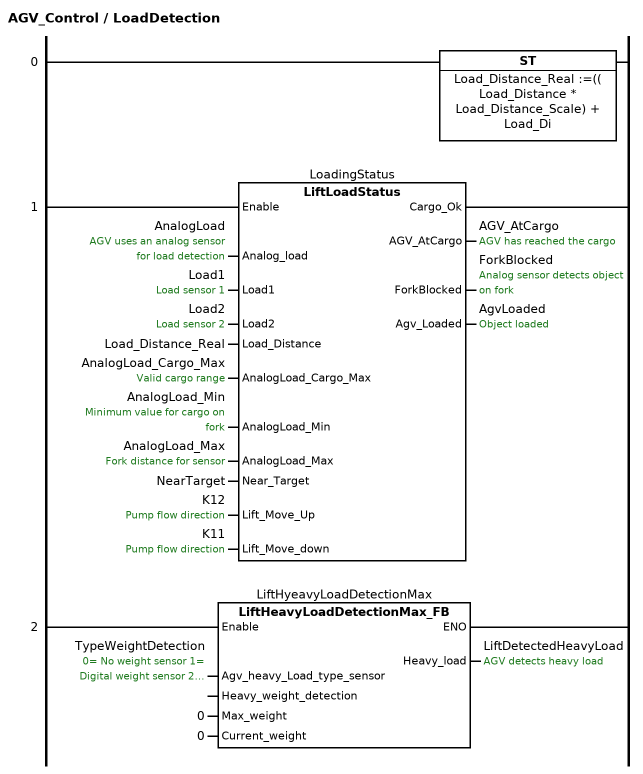
(* Rung 0 *)
Load_Distance_Real :=(( Load_Distance * Load_Distance_Scale) + Load_Distance_Offset);
(* Rung 1 *)
LoadingStatus(Enable := TRUE, Analog_load := AnalogLoad, Load1 := Load1, Load2 := Load2, Load_Distance := Load_Distance_Real, AnalogLoad_Cargo_Max := AnalogLoad_Cargo_Max, AnalogLoad_Min := AnalogLoad_Min, AnalogLoad_Max := AnalogLoad_Max, Near_Target := NearTarget, Lift_Move_Up := K12, Lift_Move_down := K11, AGV_AtCargo => AGV_AtCargo, ForkBlocked => ForkBlocked, Agv_Loaded => AgvLoaded);
(* Rung 2 *)
LiftHyeavyLoadDetectionMax(Enable := TRUE, Agv_heavy_Load_type_sensor := TypeWeightDetection, Max_weight := 0, Current_weight := 0, Heavy_load => LiftDetectedHeavyLoad);

(* Section Bufferlane: ladder, written here as Structured Text *)

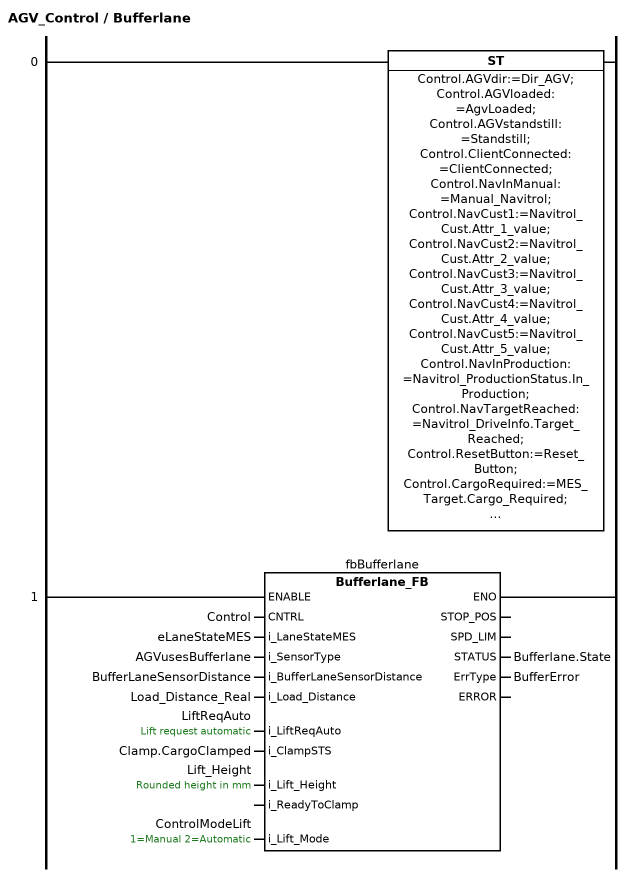
(* Rung 0 *)
Control.AGVdir:=Dir_AGV;
Control.AGVloaded:=AgvLoaded;
Control.AGVstandstill:=Standstill;
Control.ClientConnected:=ClientConnected;
Control.NavInManual:=Manual_Navitrol;
Control.NavCust1:=Navitrol_Cust.Attr_1_value;
Control.NavCust2:=Navitrol_Cust.Attr_2_value;
Control.NavCust3:=Navitrol_Cust.Attr_3_value;
Control.NavCust4:=Navitrol_Cust.Attr_4_value;
Control.NavCust5:=Navitrol_Cust.Attr_5_value;
Control.NavInProduction:=Navitrol_ProductionStatus.In_Production;
Control.NavTargetReached:=Navitrol_DriveInfo.Target_Reached;
Control.ResetButton:=Reset_Button;
Control.CargoRequired:=MES_Target.Cargo_Required;

MES_LanePickState:=Bufferlane.State.ePickSTAT;
MES_LaneDropState:=Bufferlane.State.eDropSTAT;
(* Rung 1 *)
fbBufferlane(ENABLE := TRUE, CNTRL := Control, i_LaneStateMES := eLaneStateMES, i_SensorType := AGVusesBufferlane, i_BufferLaneSensorDistance := BufferLaneSensorDistance, i_Load_Distance := Load_Distance_Real, i_LiftReqAuto := LiftReqAuto, i_ClampSTS := Clamp.CargoClamped, i_Lift_Height := Lift_Height, i_Lift_Mode := ControlModeLift, STATUS => Bufferlane.State, ErrType => BufferError);
END_PROGRAM

PROGRAM Communication
VAR
    Host : STRING[256];
    ServerPort : INT;
    Willconfig_Mqtt : MQTT\WillCnfg;
    mqttbuffer : MQTT\ClientBuffer;
    mqttclient : MQTT\MQTTClient;
    start_up : TON;
    mqttping : MQTT\MQTTPing;
    rcv_message : STRING[1986];
    rcv_topic : STRING[128];
    mqttsub : MQTT\MQTTSubscribe;
    rcv_message_mes : STRING[1986];
    rcv_topic_mes : STRING[128];
    mqttsub_mes : MQTT\MQTTSubscribe;
    rcv_message_target : STRING[1986];
    rcv_topic_target : STRING[128];
    mqttsub_target : MQTT\MQTTSubscribe;
    sendRequest : BOOL;
    mqttpublish : MQTT\MQTTPublish;
    pub_topic : STRING[128];
    act_topic : STRING[128];  (* MQTT topic for actuator commands from MES *)
    pub_message : STRING[1986];
    act_message : STRING[1986];  (* MQTT message for responding to actuator commands *)
    pub_i : UINT;
END_VAR
VAR RETAIN
    machid : STRING[20];
END_VAR
VAR
    SerialSetupDone : BOOL;  (* RS232 setup state done *)
    RS_TX_Done : BOOL;  (* Serial buffer send *)
    debug_receiveserial : BOOL;
    debug_sendserial : BOOL;
    SendSerial1 : BOOL;  (* Send serial message 1 *)
    SerialTimer_PT : TIME;  (* Cycle time *)
    SerialTimer_ET : TIME;  (* Elapsed time *)
    SerialTimer_TON : TON;
    RS_Clear_Done : BOOL;  (* Serial buffer cleared *)
    DevicePort : _sDEVICE_PORT;  (* RS232 port *)
    SerialSendDat : ARRAY[0..4] OF BYTE;  (* TX byte array *)
    SerialSendSize : UINT;  (* Amount of bytes to send *)
    SerialSendConfig : _sSERIAL_CFG;  (* Block config *)
    SerialSendOption : _sSERIAL_SEND_OPTION;  (* Transmission option *)
    RS_Abort : BOOL;  (* Halt serial communication *)
    RS_TX_Busy : BOOL;  (* Transmission in progress *)
    RS_TX_Aborted : BOOL;  (* Transmission has been aborted *)
    RS_TX_Error : BOOL;  (* Error active in serial send *)
    RS_TX_ErrorID : WORD;  (* Error ID *)
    RS232_TX : NX_SerialSend;  (* Send serial data *)
    RS_RX_Done : BOOL;  (* Serial buffer read *)
    SerialReceive : ARRAY[0..49] OF BYTE;  (* Serial message in Bytes *)
    SerialRecvSize : UINT;  (* Amount of bytes we want to read *)
    SerialRcvConfig : _sSERIAL_CFG;  (* block config *)
    SerialRcvOption : _sSERIAL_RCV_OPTION;  (* Transmission option *)
    RS_RS_Busy : BOOL;  (* Read in progress *)
    RS_RX_Aborted : BOOL;  (* Read has been aborted *)
    RS_RX_Error : BOOL;  (* Error active in serial read *)
    RS_RX_ErrorID : WORD;  (* Error ID *)
    RS_RX_Size : UINT;  (* Amount of bytes read *)
    RS232_RX : NX_SerialRcv;  (* Receive serial data from buffer *)
    debug_clearserial : BOOL;
    RS232_Clear_Busy : BOOL;  (* Buffer clearing in pogress *)
    RS232_Clear : NX_SerialBufClear;  (* Serial RXbuffer clear *)
    HandleSerialData : BOOL;  (* Apply filters and calculate distance *)
    ReceivedChecksum : BYTE;  (* Last received XOR checksum *)
    SerialOk : BOOL;  (* Checksum ok on received data *)
    SerialDataSaved : BOOL;  (* All distances and echos received ok *)
    Distances : ARRAY[0..10] OF UINT;  (* All distances from RS232 sensor *)
    Echos : ARRAY[0..10] OF UINT;  (* All echos from RS232 sensor *)
    FirstUpdateDone : BOOL;  (* Serial data has been received *)
    OverhangDetected : BOOL;  (* Overhead detection measurements within limit *)
    Overhang_ChargerOverride : BOOL;  (* AGV is aproaching the charger *)
    Overhang_PT : TIME;  (* time an object must be within bounds *)
    Overhang_ET : TIME;  (* Elapsed time *)
    Overhang_TON : TON;  (* Overhang stability timer *)
    Checksum : BYTE;  (* Calculated checksum *)
    IndexCheck : UINT;  (* index for checksum calculation *)
    NrOfBeams : UINT;  (* Amount of beams per scan *)
    Xserial : ARRAY[0..10] OF INT;  (* Calculated X values from measurements *)
    Angle : ARRAY[0..10] OF REAL;  (* Angles in radians *)
    Yserial : ARRAY[0..10] OF INT;  (* Calculated Y values from measurements *)
    IndexLimit : UINT;
    Ylimit : INT;  (* Distance the RS232 beams are allowed to go sideways *)
    Xlimit : INT;  (* Distance the RS232 beams should be able to reach towards the front *)
    PublishIndex : INT;
    MqttActRequest : BOOL;  (* Transmit update *)
    mqtt_target_publish : MQTT\MQTTPublish;
    mqttsub_palletDetection : MQTT\MQTTSubscribe;
    palletDetection_topic : STRING[128];
    rcv_message_palletDetection : STRING[1986];
    rcv_topic_palletDetection : STRING[128];
    Mqtt_client_ID : STRING[128];
    error_topic : STRING[128];
    HMI_IP_Init : BOOL;
    Host_Block1 : STRING[18];
    Host_Block2 : STRING[18];
    mqtt_test_done : BOOL;
    mqttsub_error : MQTT\MQTTSubscribe;
    mqttsub_popup : MQTT\MQTTSubscribe;
    mqttsub_warning : MQTT\MQTTSubscribe;
    popup_topic : STRING[128];
    rcv_message_error : STRING[1986];
    rcv_message_popup : STRING[1986];
    rcv_message_warning : STRING[1986];
    rcv_popup_info : STRING[128];
    rcv_topic_error : STRING[128];
    rcv_topic_warning : STRING[128];
    warning_topic : STRING[128];
    mqttsub_language : MQTT\MQTTSubscribe;
    language_topic : STRING[128];
    laneDropStateMES_topic : STRING[128];
    laneStateMES_topic : STRING[128];
    mqttsub_laneStateMES : MQTT\MQTTSubscribe;
    mqttsub_MES_BufferState : MQTT\MQTTSubscribe;
    rcv_message_laneDropStateMES : STRING[1986];
    rcv_message_laneStateMES : STRING[128];
    rcv_topic_laneDropStateMES : STRING[128];
    rcv_topic_laneStateMES : STRING[128];
END_VAR
VAR_EXTERNAL
    ClientConnected : BOOL;
    Mqtt_values : ARRAY[0..32] OF MQTTval;
    Stations_State : Node_State;
    MES_State : Node_State;
    MES_Target : MQTT_Actuator_Request_struct;
    AGVusesRS232 : BOOL;
    AGV_Init : UINT;
    Dir_Encoder1 : BOOL;
    Brake_Override_Switch : BOOL;
    Manual_ControlModeLift : BOOL;
    AGV_Docking : BOOL;
    Reset_Flag : BOOL;
    Navitrol_Tag : Navitrol_Status_TagV4_sec_struct;
    ToChargerTag : UDINT;
    ChargerTag : UDINT;
    Standstill : BOOL;
    Charge_Relay : BOOL;
END_VAR
VAR_EXTERNAL CONSTANT
    RS232_BoardID : _sOPTBOARD_ID;
END_VAR
VAR_EXTERNAL
    MachineID : INT;
    Warning_Mqtt_Client_Error : BOOL;
    MQTT_enabled : BOOL;  (* MES communication type enabled *)
    MES_PalletDetection : Palletdetection_Action;
    OptionalFieldReq : INT;
    RS232_OverhangDetected : BOOL;
    HMI_Int12 : INT;
    HMI_Int13 : INT;
    HMI_Int14 : INT;
    HMI_Int15 : INT;
    IP_Block1 : INT;
    IP_Block2 : INT;
    IP_Block3 : INT;
    IP_Block4 : INT;
    MES_Error : MQTT_Errors_struct;
    MES_Popup : MQTT_Popup_struct;
    MES_Warning : MQTT_Warnings_struct;
    HMI_Input13 : BOOL;
    HMI_Int16 : INT;
    MES_Language : INT;
    eLaneStateMES : Lane_state_MES;
    Manual_Mode : BOOL;
END_VAR
VAR
    _p1 : BOOL;
    _e2 : R_TRIG;
    _e3 : R_TRIG;
    _e4 : R_TRIG;
    _e5 : R_TRIG;
    _p6 : BOOL;
    _p7 : BOOL;
END_VAR

(* Section Client: ladder, written here as Structured Text *)

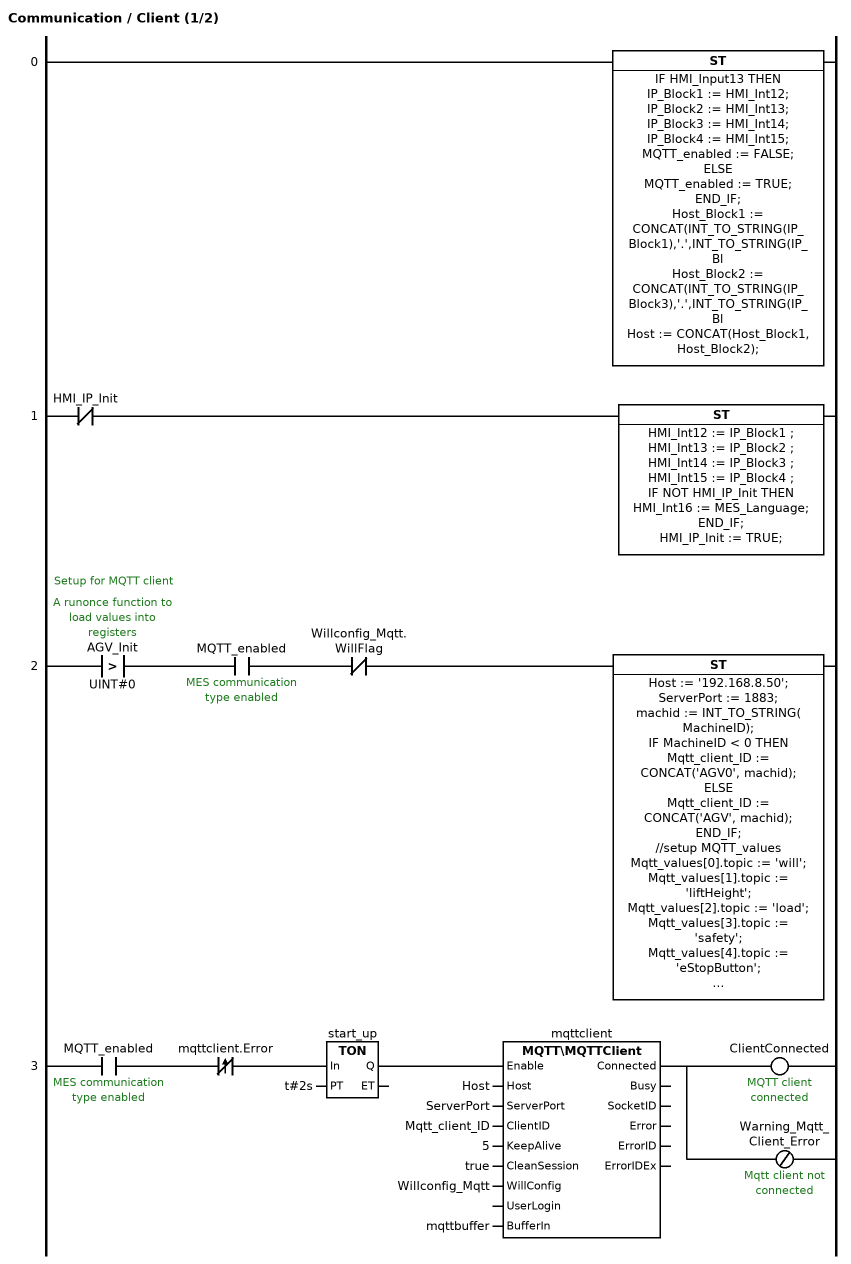
(* Rung 0 *)
IF HMI_Input13 THEN
	IP_Block1 := HMI_Int12;
	IP_Block2 := HMI_Int13;
	IP_Block3 := HMI_Int14;
	IP_Block4 := HMI_Int15;

	MQTT_enabled := FALSE;
	
ELSE
	MQTT_enabled := TRUE;
END_IF;

Host_Block1 := CONCAT(INT_TO_STRING(IP_Block1),'.',INT_TO_STRING(IP_Block2),'.');
Host_Block2 := CONCAT(INT_TO_STRING(IP_Block3),'.',INT_TO_STRING(IP_Block4));
Host := CONCAT(Host_Block1,Host_Block2);
(* Rung 1 *)
_p1 := NOT HMI_IP_Init;
IF _p1 THEN
    HMI_Int12 := IP_Block1 ;
    HMI_Int13 := IP_Block2 ;
    HMI_Int14 := IP_Block3 ;
    HMI_Int15 := IP_Block4 ;
    
    IF NOT HMI_IP_Init THEN
    	HMI_Int16 := MES_Language;
    END_IF;
    
    HMI_IP_Init := TRUE;
END_IF;
(* Rung 2: Setup for MQTT client *)
IF (AGV_Init > UINT#0) AND MQTT_enabled AND NOT Willconfig_Mqtt.WillFlag THEN
    Host := '192.168.8.50';
    ServerPort := 1883;
    machid := INT_TO_STRING(MachineID);
    IF MachineID < 0 THEN
    	Mqtt_client_ID := CONCAT('AGV0', machid);
    ELSE
    	Mqtt_client_ID := CONCAT('AGV', machid);
    END_IF;
    
    //setup MQTT_values
    Mqtt_values[0].topic := 'will';
    Mqtt_values[1].topic := 'liftHeight';
    Mqtt_values[2].topic := 'load';
    Mqtt_values[3].topic := 'safety';
    Mqtt_values[4].topic := 'eStopButton';
    Mqtt_values[5].topic := 'scanner1';
    Mqtt_values[6].topic := 'scanner2';
    Mqtt_values[7].topic := 'palletDetection/state';
    Mqtt_values[8].topic := 'docking';
    Mqtt_values[9].topic := 'manualDrive';
    Mqtt_values[10].topic := 'manualLift';
    Mqtt_values[11].topic := 'brakeRelease';
    Mqtt_values[12].topic := 'charging';
    Mqtt_values[13].topic := 'cancelRequest';
    Mqtt_values[14].topic := 'cancelConfirm';
    Mqtt_values[15].topic := 'forkCollision';
    Mqtt_values[16].topic := 'palletDetection/countedPallets';
    Mqtt_values[17].topic := 'heavyLoad';
    Mqtt_values[18].topic := 'laneDropStateAGV';
    Mqtt_values[19].topic := 'palletDetection';
    Mqtt_values[20].topic := 'errorsWarnings';
    Mqtt_values[21].topic := 'palletDetectionAngle';
    Mqtt_values[22].topic := 'popUp/operatorConfirmation';
    Mqtt_values[23].topic := 'popUp/operatorCancelation';
    Mqtt_values[24].topic := 'language';
    Mqtt_values[25].topic := 'lanePickStateAGV';
    
    //config for firstrun. required for startup
    Willconfig_Mqtt.WillTopic :=  CONCAT('agvs/',machid,'/will');
    Willconfig_Mqtt.WillMsg := 'Offline';
    Willconfig_Mqtt.WillRetain := TRUE;
    Willconfig_Mqtt.WillQoS := 0;
    Willconfig_Mqtt.WillFlag := TRUE;
    
    //Actuator values
    act_topic := CONCAT('agvs/',INT_TO_STRING(MachineID),'/target');
    palletDetection_topic := CONCAT('agvs/',INT_TO_STRING(MachineID),'/palletDetection/active');
    popup_topic:=CONCAT('agvs/',INT_TO_STRING(MachineID),'/popUp');
    language_topic:=CONCAT('agvs/',INT_TO_STRING(MachineID),'/language');
    laneStateMES_topic:=CONCAT('agvs/',INT_TO_STRING(MachineID),'/laneActionStateMES');
END_IF;
(* Rung 3 *)
_e2(CLK := mqttclient.Error);
start_up(In := MQTT_enabled AND NOT _e2.Q, PT := t#2s);
mqttclient(Enable := start_up.Q, Host := Host, ServerPort := ServerPort, ClientID := Mqtt_client_ID, KeepAlive := 5, CleanSession := true, WillConfig := Willconfig_Mqtt, BufferIn := mqttbuffer);
ClientConnected := mqttclient.Connected;
Warning_Mqtt_Client_Error := NOT mqttclient.Connected;

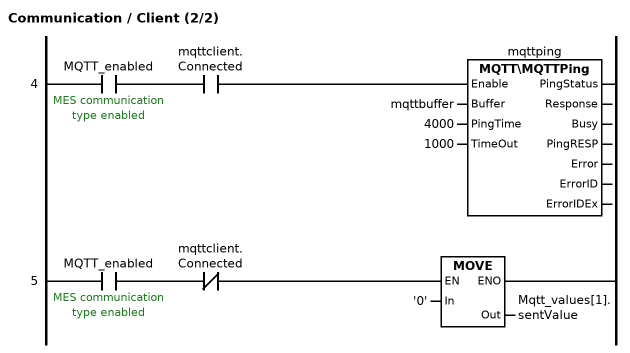
(* Rung 4 *)
mqttping(Enable := MQTT_enabled AND mqttclient.Connected, Buffer := mqttbuffer, PingTime := 4000, TimeOut := 1000);
(* Rung 5 *)
IF MQTT_enabled AND NOT mqttclient.Connected THEN Mqtt_values[1].sentValue := '0'; END_IF;

(* Section Subscribe: ladder, written here as Structured Text *)

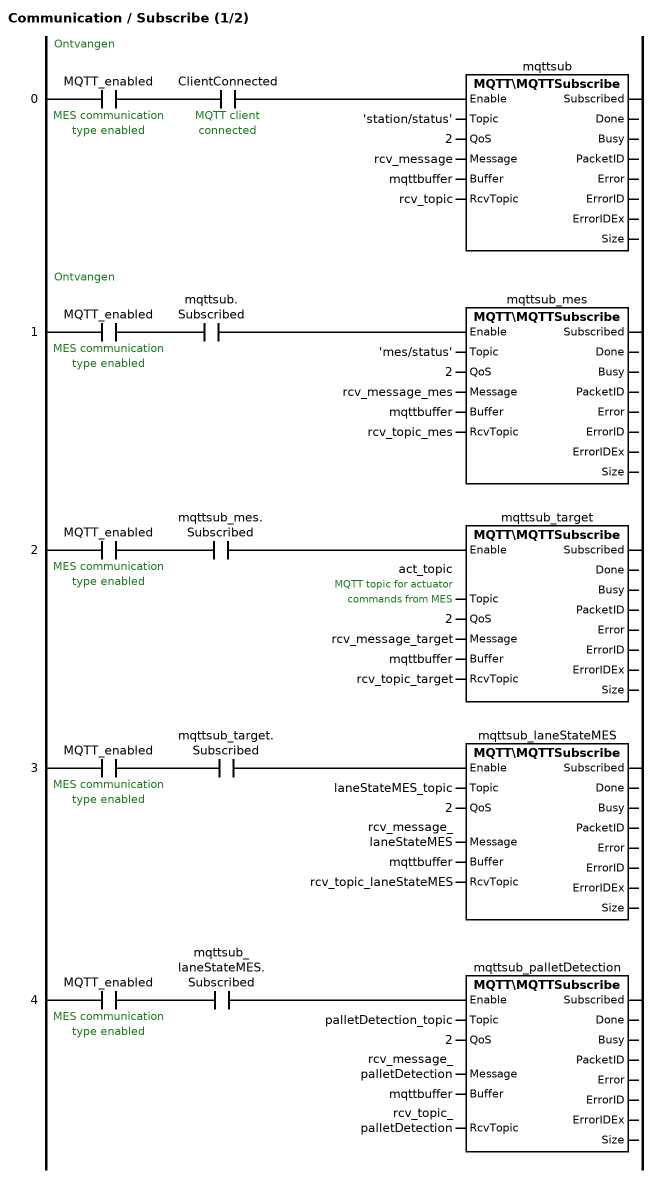
(* Rung 0: Ontvangen *)
mqttsub(Enable := MQTT_enabled AND ClientConnected, Topic := 'station/status', QoS := 2, Message := rcv_message, Buffer := mqttbuffer, RcvTopic := rcv_topic);
(* Rung 1: Ontvangen *)
mqttsub_mes(Enable := MQTT_enabled AND mqttsub.Subscribed, Topic := 'mes/status', QoS := 2, Message := rcv_message_mes, Buffer := mqttbuffer, RcvTopic := rcv_topic_mes);
(* Rung 2 *)
mqttsub_target(Enable := MQTT_enabled AND mqttsub_mes.Subscribed, Topic := act_topic, QoS := 2, Message := rcv_message_target, Buffer := mqttbuffer, RcvTopic := rcv_topic_target);
(* Rung 3 *)
mqttsub_laneStateMES(Enable := MQTT_enabled AND mqttsub_target.Subscribed, Topic := laneStateMES_topic, QoS := 2, Message := rcv_message_laneStateMES, Buffer := mqttbuffer, RcvTopic := rcv_topic_laneStateMES);
(* Rung 4 *)
mqttsub_palletDetection(Enable := MQTT_enabled AND mqttsub_laneStateMES.Subscribed, Topic := palletDetection_topic, QoS := 2, Message := rcv_message_palletDetection, Buffer := mqttbuffer, RcvTopic := rcv_topic_palletDetection);

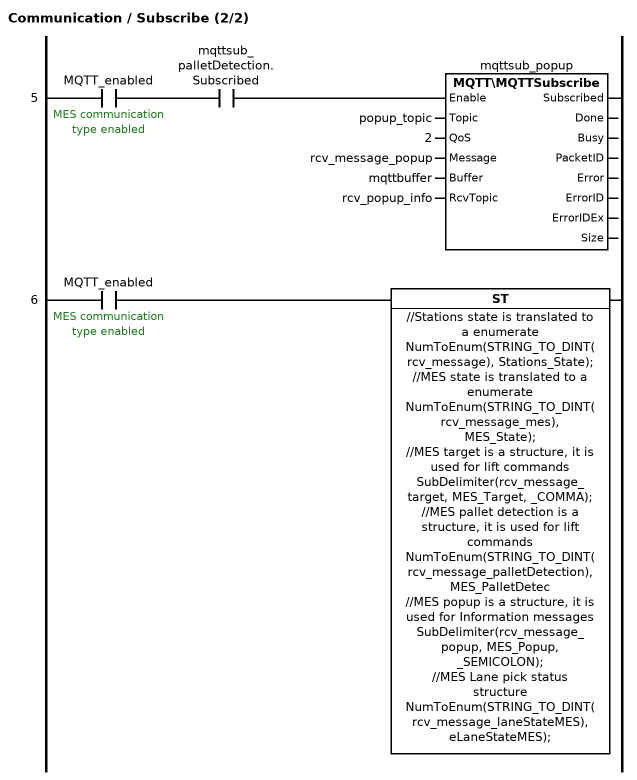
(* Rung 5 *)
mqttsub_popup(Enable := MQTT_enabled AND mqttsub_palletDetection.Subscribed, Topic := popup_topic, QoS := 2, Message := rcv_message_popup, Buffer := mqttbuffer, RcvTopic := rcv_popup_info);
(* Rung 6 *)
IF MQTT_enabled THEN
    //Stations state is translated to a enumerate
    NumToEnum(STRING_TO_DINT(rcv_message), Stations_State);
    //MES state is translated to a enumerate
    NumToEnum(STRING_TO_DINT(rcv_message_mes), MES_State);
    //MES target is a structure, it is used for lift commands
    SubDelimiter(rcv_message_target, MES_Target, _COMMA);
    //MES pallet detection is a structure, it is used for lift commands
    NumToEnum(STRING_TO_DINT(rcv_message_palletDetection), MES_PalletDetection);
    //MES popup is a structure, it is used for Information messages
    SubDelimiter(rcv_message_popup, MES_Popup, _SEMICOLON);
    //MES Lane pick status structure
    NumToEnum(STRING_TO_DINT(rcv_message_laneStateMES), eLaneStateMES);
END_IF;

(* Section Publish: ladder, written here as Structured Text *)

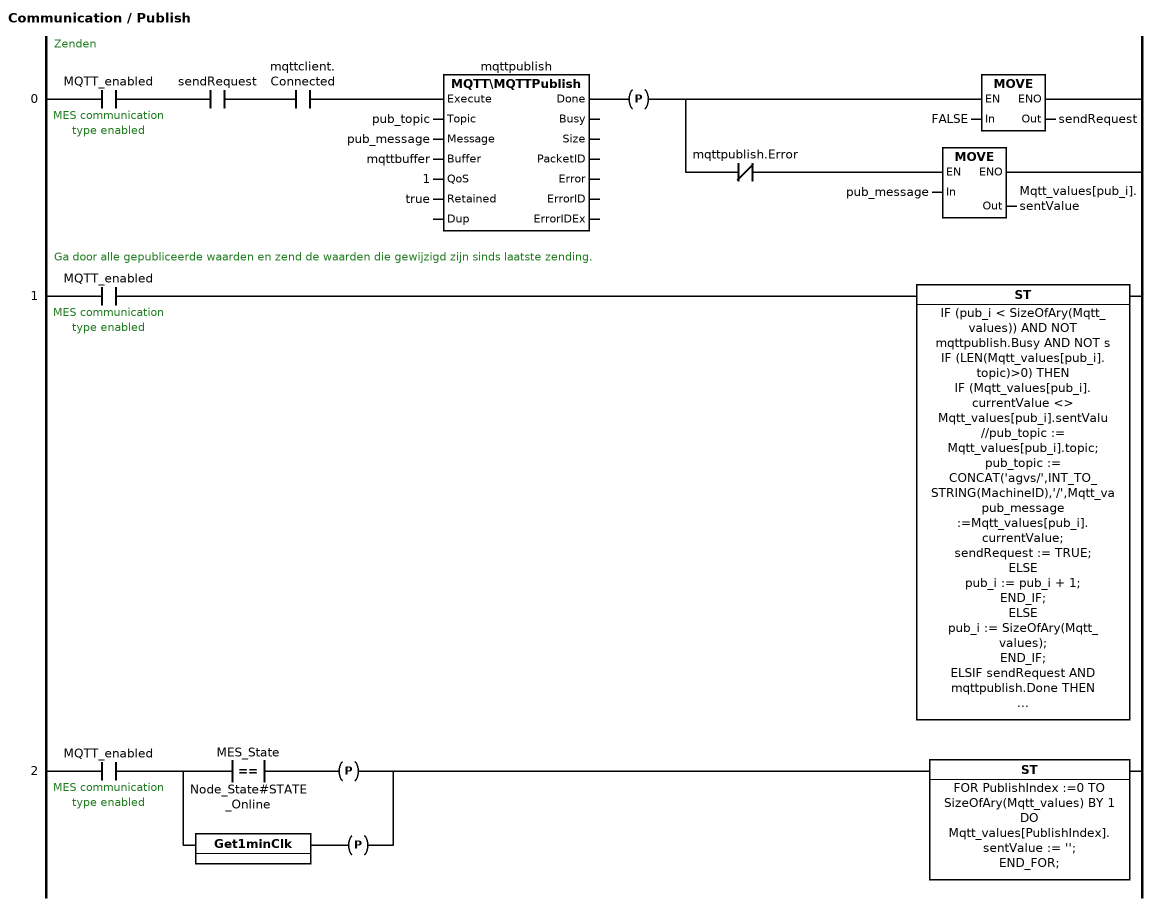
(* Rung 0: Zenden *)
mqttpublish(Execute := MQTT_enabled AND sendRequest AND mqttclient.Connected, Topic := pub_topic, Message := pub_message, Buffer := mqttbuffer, QoS := 1, Retained := true);
_e3(CLK := mqttpublish.Done);
IF _e3.Q THEN sendRequest := FALSE; END_IF;
IF _e3.Q AND NOT mqttpublish.Error THEN Mqtt_values[pub_i].sentValue := pub_message; END_IF;
(* Rung 1: Ga door alle gepubliceerde waarden en zend de waarden die gewijzigd zijn sinds laatste zending. *)
IF MQTT_enabled THEN
    IF (pub_i < SizeOfAry(Mqtt_values)) AND NOT mqttpublish.Busy AND NOT sendRequest THEN
    	IF (LEN(Mqtt_values[pub_i].topic)>0) THEN
    		IF (Mqtt_values[pub_i].currentValue <> Mqtt_values[pub_i].sentValue ) THEN
    			//pub_topic := Mqtt_values[pub_i].topic;
    			pub_topic := CONCAT('agvs/',INT_TO_STRING(MachineID),'/',Mqtt_values[pub_i].topic);
    			pub_message :=Mqtt_values[pub_i].currentValue;
    			sendRequest := TRUE;
    		ELSE
    		pub_i := pub_i + 1;
    		END_IF;
    	ELSE
    		pub_i := SizeOfAry(Mqtt_values);
    	END_IF;
    ELSIF sendRequest AND mqttpublish.Done THEN
    	sendRequest := FALSE;
    	Mqtt_values[pub_i].sentValue := pub_message;
    END_IF;
    IF (pub_i >= SizeOfAry(Mqtt_values)) THEN
    	pub_i := 0;
    END_IF;
END_IF;
(* Rung 2 *)
_e4(CLK := MQTT_enabled AND (MES_State = Node_State#STATE_Online));
_e5(CLK := MQTT_enabled AND Get1minClk());
IF _e4.Q OR _e5.Q THEN
    FOR PublishIndex :=0 TO SizeOfAry(Mqtt_values) BY 1 DO
    	Mqtt_values[PublishIndex].sentValue := '';
    END_FOR;
END_IF;

(* Section RS232: ladder, written here as Structured Text *)

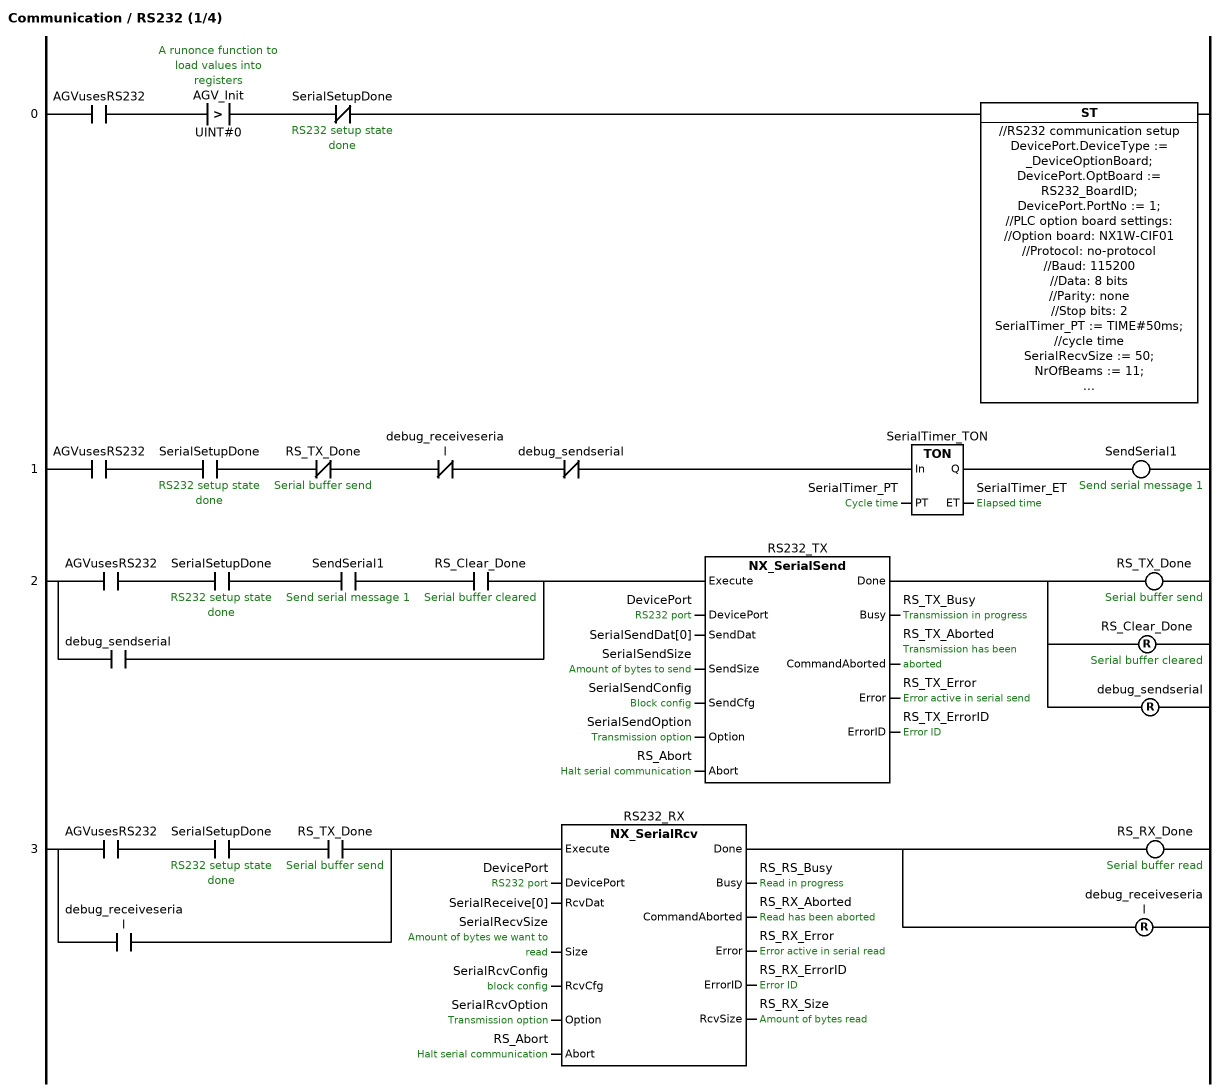
(* Rung 0 *)
IF AGVusesRS232 AND (AGV_Init > UINT#0) AND NOT SerialSetupDone THEN
    //RS232 communication setup
    DevicePort.DeviceType := _DeviceOptionBoard;
    DevicePort.OptBoard := RS232_BoardID;
    DevicePort.PortNo := 1;
    
    //PLC option board settings:
    //Option board: NX1W-CIF01
    //Protocol: no-protocol
    //Baud: 115200
    //Data: 8 bits
    //Parity: none
    //Stop bits: 2
    
    SerialTimer_PT := TIME#50ms;	//cycle time
    SerialRecvSize := 50;
    NrOfBeams := 11;
    Ylimit := 600; //distance in mm
    Xlimit := 2000; //distance in mm
    Overhang_PT := TIME#100ms;  //time an object must be in limit area until waring becomes active
    
    //TX settings
    SerialSendSize := 5;							//we send 5 bytes in total
    SerialSendOption.SendDelay := 0;	//minimal delay in transmission
    
    //Fill (Default) TX data
    SerialSendDat[0] := BYTE#222;	//0xDE = sender
    SerialSendDat[1] := BYTE#1;		//0x01 = receiver
    SerialSendDat[2] := BYTE#5;		//0x05 = amount of bytes
    SerialSendDat[3] := BYTE#89;	//0x59 = command (read)
    SerialSendDat[4] := BYTE#131;	//0x83 = XOR checksum
    
    //fill angle per beam (lookup table)
    Angle[0] := DegToRad(REAL#40);
    Angle[1] := DegToRad(REAL#32);
    Angle[2] := DegToRad(REAL#24);
    Angle[3] := DegToRad(REAL#16);
    Angle[4] := DegToRad(REAL#8);
    Angle[5] := DegToRad(REAL#0);
    Angle[6] := DegToRad(REAL#8);
    Angle[7] := DegToRad(REAL#16);
    Angle[8] := DegToRad(REAL#24);
    Angle[9] := DegToRad(REAL#32);
    Angle[10] := DegToRad(REAL#40);
    
    SerialSetupDone := TRUE;
    RS_Clear_Done := TRUE;
END_IF;
(* Rung 1 *)
SerialTimer_TON(In := AGVusesRS232 AND SerialSetupDone AND NOT RS_TX_Done AND NOT debug_receiveserial AND NOT debug_sendserial, PT := SerialTimer_PT, ET => SerialTimer_ET);
SendSerial1 := SerialTimer_TON.Q;
(* Rung 2 *)
RS232_TX(Execute := (AGVusesRS232 AND SerialSetupDone AND SendSerial1 AND RS_Clear_Done) OR debug_sendserial, DevicePort := DevicePort, SendDat := SerialSendDat[0], SendSize := SerialSendSize, SendCfg := SerialSendConfig, Option := SerialSendOption, Abort := RS_Abort, Busy => RS_TX_Busy, CommandAborted => RS_TX_Aborted, Error => RS_TX_Error, ErrorID => RS_TX_ErrorID);
RS_TX_Done := RS232_TX.Done;
IF RS232_TX.Done THEN
    RS_Clear_Done := FALSE;
    debug_sendserial := FALSE;
END_IF;
(* Rung 3 *)
RS232_RX(Execute := (AGVusesRS232 AND SerialSetupDone AND RS_TX_Done) OR debug_receiveserial, DevicePort := DevicePort, RcvDat := SerialReceive[0], Size := SerialRecvSize, RcvCfg := SerialRcvConfig, Option := SerialRcvOption, Abort := RS_Abort, Busy => RS_RS_Busy, CommandAborted => RS_RX_Aborted, Error => RS_RX_Error, ErrorID => RS_RX_ErrorID, RcvSize => RS_RX_Size);
RS_RX_Done := RS232_RX.Done;
IF RS232_RX.Done THEN debug_receiveserial := FALSE; END_IF;

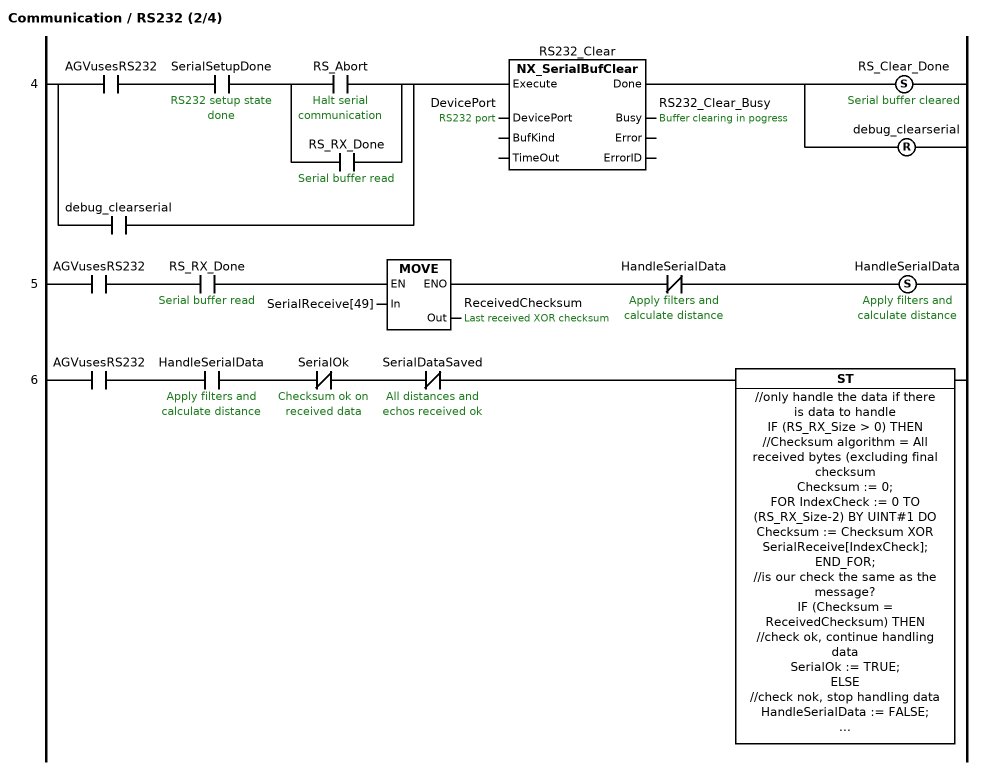
(* Rung 4 *)
RS232_Clear(Execute := (AGVusesRS232 AND SerialSetupDone AND (RS_Abort OR RS_RX_Done)) OR debug_clearserial, DevicePort := DevicePort, Busy => RS232_Clear_Busy);
IF RS232_Clear.Done THEN
    RS_Clear_Done := TRUE;
    debug_clearserial := FALSE;
END_IF;
(* Rung 5 *)
IF AGVusesRS232 AND RS_RX_Done THEN ReceivedChecksum := SerialReceive[49]; END_IF;
IF AGVusesRS232 AND RS_RX_Done AND NOT HandleSerialData THEN HandleSerialData := TRUE; END_IF;
(* Rung 6 *)
_p6 := AGVusesRS232 AND HandleSerialData AND NOT SerialOk AND NOT SerialDataSaved;
IF _p6 THEN
    //only handle the data if there is data to handle
    IF (RS_RX_Size > 0) THEN
    	//Checksum algorithm = All received bytes (excluding final checksum byte) must be XOR
    	Checksum := 0;
    	FOR IndexCheck := 0 TO (RS_RX_Size-2) BY UINT#1 DO
    		Checksum := Checksum XOR SerialReceive[IndexCheck];
    	END_FOR;
    	//is our check the same as the message?
    	IF (Checksum = ReceivedChecksum) THEN
    		//check ok, continue handling data
    		SerialOk := TRUE;
    	ELSE
    		//check nok, stop handling data
    		HandleSerialData := FALSE;
    	END_IF;
    ELSE
    	//no data, stop handling data
    	HandleSerialData := FALSE;
    END_IF;
    	
END_IF;

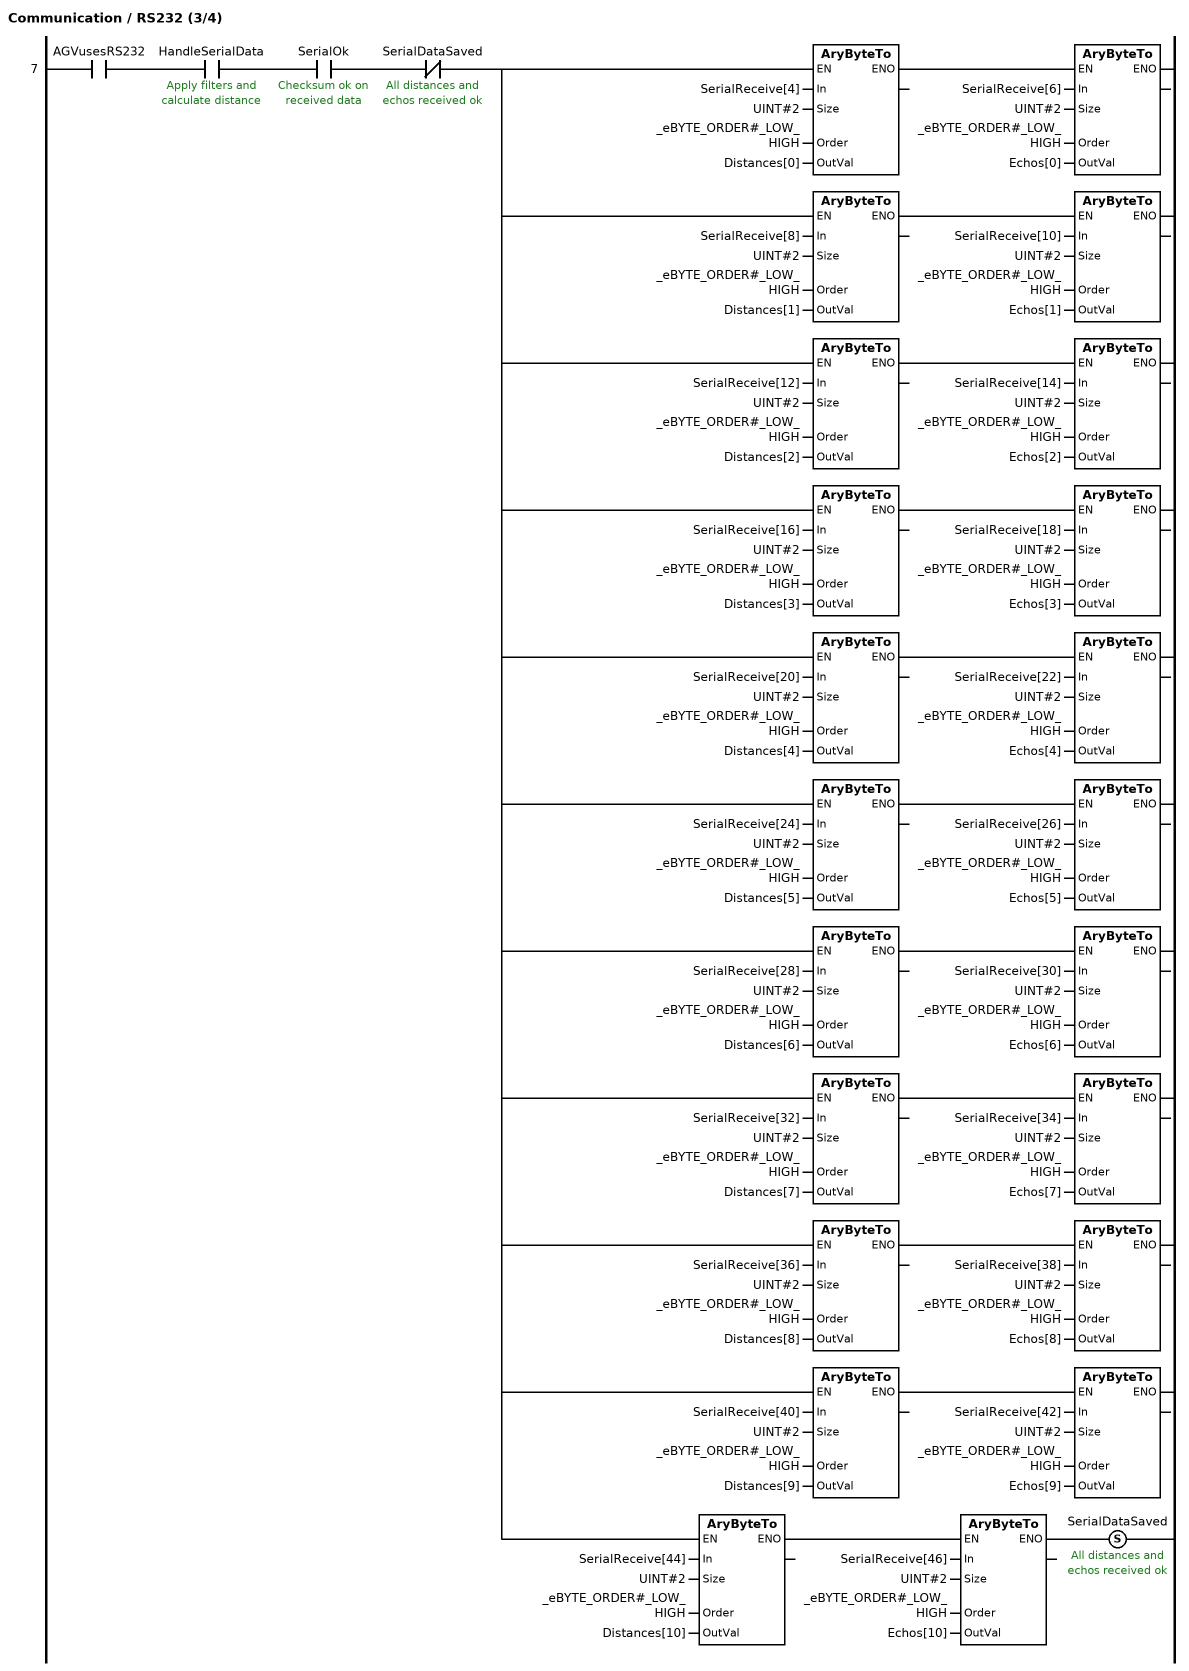
(* Rung 7 *)
_p7 := AGVusesRS232 AND HandleSerialData AND SerialOk AND NOT SerialDataSaved;
IF _p7 THEN
    AryByteTo(In := SerialReceive[4], Size := UINT#2, Order := _eBYTE_ORDER#_LOW_HIGH, OutVal := Distances[0]);
    AryByteTo(In := SerialReceive[6], Size := UINT#2, Order := _eBYTE_ORDER#_LOW_HIGH, OutVal := Echos[0]);
    AryByteTo(In := SerialReceive[8], Size := UINT#2, Order := _eBYTE_ORDER#_LOW_HIGH, OutVal := Distances[1]);
    AryByteTo(In := SerialReceive[10], Size := UINT#2, Order := _eBYTE_ORDER#_LOW_HIGH, OutVal := Echos[1]);
    AryByteTo(In := SerialReceive[12], Size := UINT#2, Order := _eBYTE_ORDER#_LOW_HIGH, OutVal := Distances[2]);
    AryByteTo(In := SerialReceive[14], Size := UINT#2, Order := _eBYTE_ORDER#_LOW_HIGH, OutVal := Echos[2]);
    AryByteTo(In := SerialReceive[16], Size := UINT#2, Order := _eBYTE_ORDER#_LOW_HIGH, OutVal := Distances[3]);
    AryByteTo(In := SerialReceive[18], Size := UINT#2, Order := _eBYTE_ORDER#_LOW_HIGH, OutVal := Echos[3]);
    AryByteTo(In := SerialReceive[20], Size := UINT#2, Order := _eBYTE_ORDER#_LOW_HIGH, OutVal := Distances[4]);
    AryByteTo(In := SerialReceive[22], Size := UINT#2, Order := _eBYTE_ORDER#_LOW_HIGH, OutVal := Echos[4]);
    AryByteTo(In := SerialReceive[24], Size := UINT#2, Order := _eBYTE_ORDER#_LOW_HIGH, OutVal := Distances[5]);
    AryByteTo(In := SerialReceive[26], Size := UINT#2, Order := _eBYTE_ORDER#_LOW_HIGH, OutVal := Echos[5]);
    AryByteTo(In := SerialReceive[28], Size := UINT#2, Order := _eBYTE_ORDER#_LOW_HIGH, OutVal := Distances[6]);
    AryByteTo(In := SerialReceive[30], Size := UINT#2, Order := _eBYTE_ORDER#_LOW_HIGH, OutVal := Echos[6]);
    AryByteTo(In := SerialReceive[32], Size := UINT#2, Order := _eBYTE_ORDER#_LOW_HIGH, OutVal := Distances[7]);
    AryByteTo(In := SerialReceive[34], Size := UINT#2, Order := _eBYTE_ORDER#_LOW_HIGH, OutVal := Echos[7]);
    AryByteTo(In := SerialReceive[36], Size := UINT#2, Order := _eBYTE_ORDER#_LOW_HIGH, OutVal := Distances[8]);
    AryByteTo(In := SerialReceive[38], Size := UINT#2, Order := _eBYTE_ORDER#_LOW_HIGH, OutVal := Echos[8]);
    AryByteTo(In := SerialReceive[40], Size := UINT#2, Order := _eBYTE_ORDER#_LOW_HIGH, OutVal := Distances[9]);
    AryByteTo(In := SerialReceive[42], Size := UINT#2, Order := _eBYTE_ORDER#_LOW_HIGH, OutVal := Echos[9]);
    AryByteTo(In := SerialReceive[44], Size := UINT#2, Order := _eBYTE_ORDER#_LOW_HIGH, OutVal := Distances[10]);
    AryByteTo(In := SerialReceive[46], Size := UINT#2, Order := _eBYTE_ORDER#_LOW_HIGH, OutVal := Echos[10]);
    SerialDataSaved := TRUE;
END_IF;

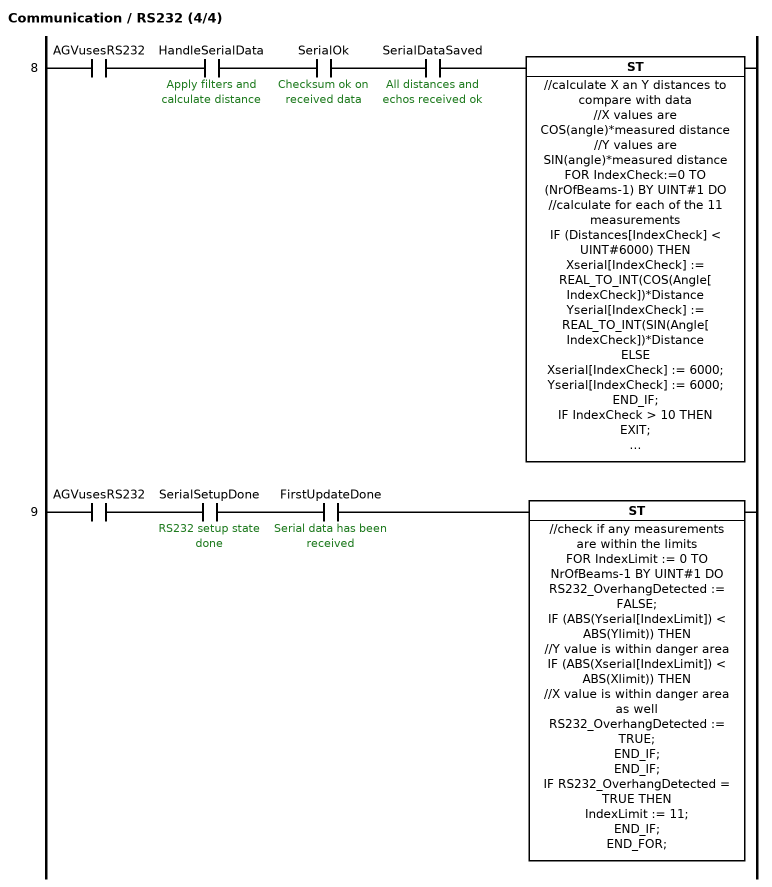
(* Rung 8 *)
IF AGVusesRS232 AND HandleSerialData AND SerialOk AND SerialDataSaved THEN
    //calculate X an Y distances to compare with data
    //X values are COS(angle)*measured distance
    //Y values are SIN(angle)*measured distance
    FOR IndexCheck:=0 TO (NrOfBeams-1) BY UINT#1 DO
    	//calculate for each of the 11 measurements
    	IF (Distances[IndexCheck] < UINT#6000) THEN
    		Xserial[IndexCheck] := REAL_TO_INT(COS(Angle[IndexCheck])*Distances[IndexCheck]);
    		Yserial[IndexCheck] := REAL_TO_INT(SIN(Angle[IndexCheck])*Distances[IndexCheck]);
    	ELSE
    		Xserial[IndexCheck] := 6000;
    		Yserial[IndexCheck] := 6000;
    	END_IF;
    	IF IndexCheck > 10 THEN
    		EXIT;
    	END_IF;
    END_FOR;
    
    //Checks done
    SerialDataSaved := FALSE;
    SerialOk := FALSE;
    HandleSerialData := FALSE;
    FirstUpdateDone := TRUE;
END_IF;
(* Rung 9 *)
IF AGVusesRS232 AND SerialSetupDone AND FirstUpdateDone THEN
    //check if any measurements are within the limits
    FOR IndexLimit := 0 TO NrOfBeams-1 BY UINT#1 DO
    	RS232_OverhangDetected := FALSE;
    	IF (ABS(Yserial[IndexLimit]) < ABS(Ylimit)) THEN
    		//Y value is within danger area
    		IF (ABS(Xserial[IndexLimit]) < ABS(Xlimit)) THEN
    			//X value is within danger area as well
    			RS232_OverhangDetected := TRUE;
    		END_IF;
    	END_IF;
    	IF RS232_OverhangDetected = TRUE THEN
    		IndexLimit := 11;
    	END_IF;
    END_FOR;
END_IF;
END_PROGRAM

PROGRAM Manual_control
VAR
    AnalogFwdRevInput : INT := 0;  (* Combined input from both F/R channels *)
END_VAR
VAR CONSTANT
    CenterCounts : INT := 1000;  (* 2,5V on -4000/4000 counts *)
    AnalogMaxFwdCounts : INT := 2000;  (* Maximum counts when joystick max forward *)
    AnalogMaxLeftCounts : INT := 0;  (* Maximum counts when joystick max left *)
    AnalogMaxRevCounts : INT := 0000;  (* Minimum counts when joystick max reverse *)
    AnalogMaxRightCounts : INT := 2000;  (* Minimum counts when joystick max right *)
END_VAR
VAR
    PercentFwdRev : INT := 0;  (* Percentage in forward/reverse (-100=max rev, 100 = max fwd) *)
    PercentLeftRight : INT := 0;  (* Percentage in left/right (-100=max left, 100=max right) *)
    AnalogLeftRightInput : INT := 0;
    RM_FR1Avg : INT := 0;  (* Average value of RM_FR1 channel *)
    alpha : INT := 10;  (* alpha = between 0 and 100, for averaging *)
    RM_LR1Avg : INT := 0;  (* Average value of RM_LR1 channel *)
    RM_CenterAvg : INT := 0;  (* Average value of RM_Center channel *)
    ManualConnect : SktTCPConnect;
    ManualSocket : _sSOCKET;
    ManualSend : SktTCPSend;
    payload : ARRAY[0..150] OF BYTE := [16#50,16#4f,16#53,16#54,16#20,16#2f,16#72,16#65,16#6d,16#6f,16#74,16#65,16#5f,16#63,16#6f,16#6e,16#74,16#72,16#6f,16#6c,16#3f,16#78,16#3d,16#30,16#2e,16#30,16#30,16#30,16#26,16#79,16#3d,16#30,16#2e,16#30,16#30,16#30,16#26,16#74,16#65,16#61,16#63,16#68,16#3d,16#30,16#26,16#6d,16#61,16#6e,16#75,16#61,16#6c,16#3d,16#31,16#26,16#66,16#61,16#73,16#74,16#3d,16#31,16#26,16#67,16#65,16#74,16#5f,16#63,16#6f,16#6e,16#74,16#72,16#6f,16#6c,16#3d,16#30,16#26,16#6f,16#6d,16#6e,16#69,16#5f,16#74,16#79,16#70,16#65,16#3d,16#32,16#26,16#6f,16#6d,16#6e,16#69,16#5f,16#66,16#6f,16#72,16#77,16#3d,16#31,16#20,16#48,16#54,16#54,16#50,16#2f,16#31,16#2e,16#31,16#0d,16#0a,16#48,16#6f,16#73,16#74,16#3a,16#20,16#31,16#39,16#32,16#2e,16#31,16#36,16#38,16#2e,16#31,16#32,16#37,16#2e,16#31,16#0d,16#0a,16#43,16#6f,16#6e,16#74,16#65,16#6e,16#74,16#2d,16#4c,16#65,16#6e,16#67,16#74,16#68,16#3a,16#20,16#30,16#0d,16#0a,16#0d,16#0a];
    WebPayload : ARRAY[0..250] OF BYTE;
    ASCII : ARRAY[0..9] OF BYTE := [16#30, 16#31, 16#32, 16#33, 16#34, 16#35, 16#36, 16#37, 16#38, 16#39];
    X_ABS : USINT;
    Y_ABS : USINT;
    ManualDisconnect : SktClose;
    ManualConnected : BOOL;  (* Connection to Navitrol made *)
    Sendsize : UINT;  (* amount of bytes to send *)
    Manual_Init : INT;  (* run once *)
    ManualRecv : SktTCPRcv;
    Recv_Payload : ARRAY[0..999] OF BYTE;
    Recv_Bytes : UINT;  (* Amount of bytes from buffer *)
    Got_Manual : BOOL;  (* received data *)
    Recv_String : STRING[500];
    Data_Index : UINT;
    TestByte : BYTE;
    Data_Start : STRING[9];
    debug_ButtonPressed : BOOL;
    Byte_Order : _eBYTE_ORDER := _LOW_HIGH;
    Result : UINT;
    String_Input : STRING[24];
    Got_Manual_String : BOOL;  (* Collected data *)
    Web_Feedback : Webinterface_Reply_struct;
    PLC_IP : STRING[15] := '192.168.127.2';
    debug_NEascii : BOOL;
    debug_EQascii : BOOL;
    GetToken0 : GetToken;
    TestToken : ARRAY[0..4] OF BYTE;
    Manual_Clk : BOOL;  (* debug variable *)
    Process_Manual_String : BOOL;  (* Data ready for handling *)
    Recv_Data : STRING[500];
    ManualStatus : SktGetTCPStatus;
    ManualSocket_Status : _eCONNECTION_STATE;  (* status at last send *)
    Skt_State_Closed : _eCONNECTION_STATE := _CLOSED;
    ManualClearBuffer : SktClearBuf;
    KeepAliveTON : TON;
    Keepalive_PT : TIME := 150ms;  (* time until connection is reset *)
    Keepalive_ET : TIME;  (* elapsed time *)
    ManualDisconnect0 : SktClose;
    ManualConnect0 : SktTCPConnect;
    ManualReconnect : BOOL;
    ResetAliveTON : TON;
    Skt_State_Closing : _eCONNECTION_STATE := _CLOSE_WAIT;
    String_Index : INT;
    ResetTON : TON;
    Manual_Reset_PT : TIME := 250ms;  (* time for reset *)
    Manual_Reset_ET : TIME;
    ManualTOF : TOF;
    KeepOff_PT : TIME := 50ms;  (* Reset time *)
    KeepOff_ET : TIME;  (* elapsed time *)
    GetToken1 : GetToken;
    GetToken2 : GetToken;
END_VAR
VAR_EXTERNAL
    RM_FR1 : INT;
    RM_Center : INT;
    RM_LR1 : INT;
    IPC_Driving_active : BOOL;
    IPC_Driving_x : INT;
    IPC_Driving_y : INT;
    RM_Switch : INT;
    Manual_ControlModeLift : BOOL;  (* Switch or HMI manual *)
    RemoteButtonPressed : BOOL;  (* Joystick button is pressed *)
    AGVhasHandheld : BOOL;
    Navitrol_status : Navitrol_Status_Struct;
    RM_Dwn : INT;
    RM_Up : INT;
    Remote_Present : BOOL;  (* Remote present and ok *)
    HMI_Input10 : BOOL;
    Rm_ManUp : BOOL;
    Rm_ManDown : BOOL;
    Error_Remote : BOOL;  (* Center tap voltage too low, no remote connected *)
    Navitrol_gen : Navitrol_Status_General_Sec_Struct;
    Update_Navitrol : BOOL;
    AGV_Init : UINT;
    Charge_Relay : BOOL;
    TCPReady : BOOL;
    Manual_Mode : BOOL;  (* Switch or HMI manual *)
END_VAR
VAR
    _e1 : R_TRIG;
    _e2 : F_TRIG;
    _e3 : R_TRIG;
    _p4 : BOOL;
    _e5 : R_TRIG;
    _e6 : F_TRIG;
    _e7 : R_TRIG;
    _e8 : F_TRIG;
    _e9 : F_TRIG;
    _p10 : BOOL;
    _p11 : BOOL;
    _p12 : BOOL;
    _p13 : BOOL;
END_VAR

(* Section ManualControl: ladder, written here as Structured Text *)

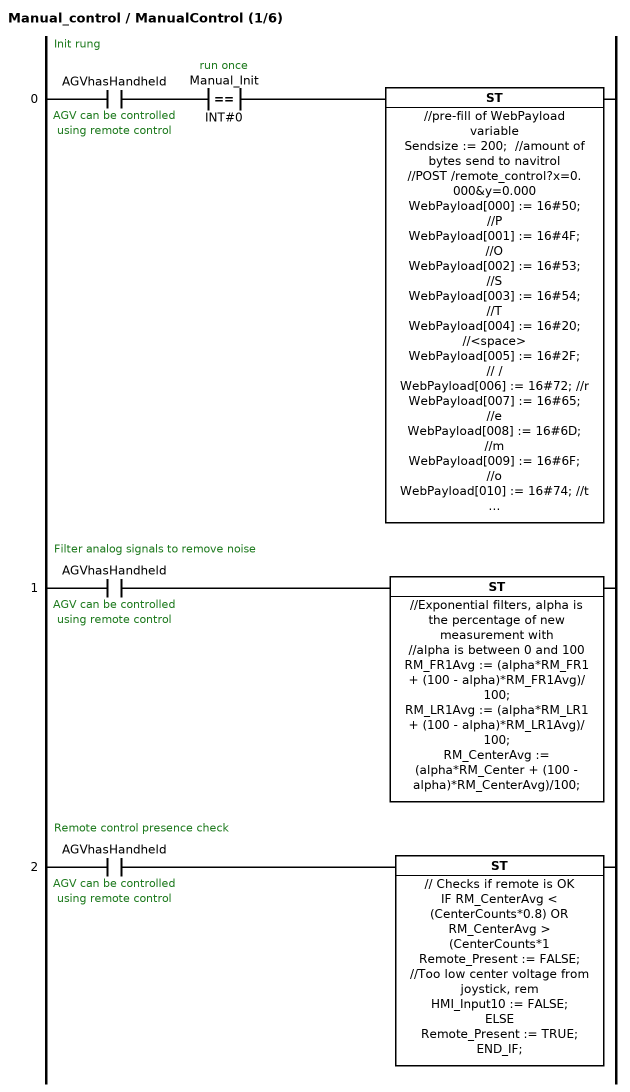
(* Rung 0: Init rung *)
IF AGVhasHandheld AND (Manual_Init = INT#0) THEN
    //pre-fill of WebPayload variable
    Sendsize := 200;	//amount of bytes send to navitrol
    //POST /remote_control?x=0.000&y=0.000
    WebPayload[000] := 16#50;	//P
    WebPayload[001] := 16#4F;		//O
    WebPayload[002] := 16#53;	//S
    WebPayload[003] := 16#54;	//T
    WebPayload[004] := 16#20;	//<space>
    WebPayload[005] := 16#2F;		// /
    WebPayload[006] := 16#72;	//r
    WebPayload[007] := 16#65;	//e
    WebPayload[008] := 16#6D;	//m
    WebPayload[009] := 16#6F;		//o
    WebPayload[010] := 16#74;	//t
    WebPayload[011] := 16#65;	//e
    WebPayload[012] := 16#5F;		//_
    WebPayload[013] := 16#63;	//c
    WebPayload[014] := 16#6F;		//o
    WebPayload[015] := 16#6E;	//n
    WebPayload[016] := 16#74;	//t
    WebPayload[017] := 16#72;	//r
    WebPayload[018] := 16#6F;		//o
    WebPayload[019] := 16#6C;	//l
    WebPayload[020] := 16#3F;		//?
    WebPayload[021] := 16#78;	//x
    WebPayload[022] := 16#3D;	//=
    WebPayload[023] := ASCII[0];	//joystick value (4 bytes)
    WebPayload[024] := 16#2E;	//.
    WebPayload[025] := ASCII[0];	//0
    WebPayload[026] := ASCII[0];	//0
    WebPayload[027] := ASCII[0];	//0
    WebPayload[028] := 16#26;	//&
    WebPayload[029] := 16#79;	//y
    WebPayload[030] := 16#3D;	//=
    WebPayload[031] := ASCII[0];	//joystick value (4 bytes)
    WebPayload[032] := 16#2E;	//.
    WebPayload[033] := ASCII[0];	//0
    WebPayload[034] := ASCII[0];	//0
    WebPayload[035] := ASCII[0];	//0
    //&teach=0
    WebPayload[036] := 16#26;	//&
    WebPayload[037] := 16#74;	//t
    WebPayload[038] := 16#65;	//e
    WebPayload[039] := 16#61;	//a
    WebPayload[040] := 16#63;	//c
    WebPayload[041] := 16#68;	//h
    WebPayload[042] := 16#3D;	//=
    WebPayload[043] := ASCII[0];	//teach ControlModeLift on/off (1 byte)
    //&manual=1
    WebPayload[044] := 16#26;	//&
    WebPayload[045] := 16#6D;	//m
    WebPayload[046] := 16#61;	//a
    WebPayload[047] := 16#6E;	//n
    WebPayload[048] := 16#75;	//u
    WebPayload[049] := 16#61;	//a
    WebPayload[050] := 16#6C;	//l
    WebPayload[051] := 16#3D;	//=
    WebPayload[052] := ASCII[0];	//manual control on/off (1 byte)
    //&fast=0
    WebPayload[053] := 16#26;	//&
    WebPayload[054] := 16#66;	//f
    WebPayload[055] := 16#61;	//a
    WebPayload[056] := 16#73;	//s
    WebPayload[057] := 16#74;	//t
    WebPayload[058] := 16#3D;	//=
    WebPayload[059] := ASCII[0];	//unkown value (1 byte)
    //&get_control=0
    WebPayload[060] := 16#26;	//&
    WebPayload[061] := 16#67;	//g
    WebPayload[062] := 16#65;	//e
    WebPayload[063] := 16#74;	//t
    WebPayload[064] := 16#5F;		//_
    WebPayload[065] := 16#63;	//c
    WebPayload[066] := 16#6F;		//o
    WebPayload[067] := 16#6E;	//n
    WebPayload[068] := 16#74;	//t
    WebPayload[069] := 16#72;	//r
    WebPayload[070] := 16#6F;		//o
    WebPayload[071] := 16#6C;	//l
    WebPayload[072] := 16#3D;	//=
    WebPayload[073] := ASCII[0];	//request to be controller (1 byte)
    //&omni_type=2
    WebPayload[074] := 16#26;	//&
    WebPayload[075] := 16#6F;		//o
    WebPayload[076] := 16#6D;	//m
    WebPayload[077] := 16#6E;	//n
    WebPayload[078] := 16#69;	//i
    WebPayload[079] := 16#5F;		//_
    WebPayload[080] := 16#74;	//t
    WebPayload[081] := 16#79;	//y
    WebPayload[082] := 16#70;	//p
    WebPayload[083] := 16#65;	//e
    WebPayload[084] := 16#3D;	//=
    WebPayload[085] := ASCII[2];	//unkown value (1 byte)
    //&omni_forw=1
    WebPayload[086] := 16#26;	//&
    WebPayload[087] := 16#6F;		//o
    WebPayload[088] := 16#6D;	//m
    WebPayload[089] := 16#6E;	//n
    WebPayload[090] := 16#69;	//i
    WebPayload[091] := 16#5F;		//_
    WebPayload[092] := 16#66;	//f
    WebPayload[093] := 16#6F;		//o
    WebPayload[094] := 16#72;	//r
    WebPayload[095] := 16#77;	//w
    WebPayload[096] := 16#3D;	//=
    WebPayload[097] := ASCII[1];	//unknown value (1 byte)
    //&token=00000
    WebPayload[098] := 16#26;	//&
    WebPayload[099] := 16#74;	//t
    WebPayload[100] := 16#6F;		//o
    WebPayload[101] := 16#6B;	//k
    WebPayload[102] := 16#65;	//e
    WebPayload[103] := 16#6E;	//n
    WebPayload[104] := 16#3D;	//=
    WebPayload[105] := ASCII[0];	//identifier (5 bytes)
    WebPayload[106] := ASCII[0];	//0
    WebPayload[107] := ASCII[0];	//0
    WebPayload[108] := ASCII[0];	//0
    WebPayload[109] := ASCII[0];	//0
    //&loadunload=0
    WebPayload[110] := 16#26;	//&
    WebPayload[111] := 16#6C;	//l
    WebPayload[112] := 16#6F;		//o
    WebPayload[113] := 16#61;	//a
    WebPayload[114] := 16#64;	//d
    WebPayload[115] := 16#75;	//u
    WebPayload[116] := 16#6E;	//n
    WebPayload[117] := 16#6C;	//l
    WebPayload[118] := 16#6F;		//o
    WebPayload[119] := 16#61;	//a
    WebPayload[120] := 16#64;	//d
    WebPayload[121] := 16#3D;	//=
    WebPayload[122] := ASCII[0];	//0
    //<space>HTTP/1.1<cr><nl>
    WebPayload[123] := 16#20;	//<space>
    WebPayload[124] := 16#48;	//H
    WebPayload[125] := 16#54;	//T
    WebPayload[126] := 16#54;	//T
    WebPayload[127] := 16#50;	//P
    WebPayload[128] := 16#2F	;	// /
    WebPayload[129] := ASCII[1];	//1
    WebPayload[130] := 16#2E;	//.
    WebPayload[131] := ASCII[1];	//1
    WebPayload[132] := 16#0D;	//<cr>
    WebPayload[133] := 16#0A;	//<nl>
    //Host:<space>192.168.127.1<cr><nl>
    WebPayload[134] := 16#48;	//H
    WebPayload[135] := 16#6F;		//o
    WebPayload[136] := 16#73;	//s
    WebPayload[137] := 16#74;	//t
    WebPayload[138] := 16#3A;	//:
    WebPayload[139] := 16#20;	//<space>
    WebPayload[140] := ASCII[1];	//1
    WebPayload[141] := ASCII[9];	//9
    WebPayload[142] := ASCII[2];	//2
    WebPayload[143] := 16#2E;	//.
    WebPayload[144] := ASCII[1];	//1
    WebPayload[145] := ASCII[6];	//6
    WebPayload[146] := ASCII[8];	//8
    WebPayload[147] := 16#2E;	//.
    WebPayload[148] := ASCII[1];	//1
    WebPayload[149] := ASCII[2];	//2
    WebPayload[150] := ASCII[7];	//7
    WebPayload[151] := 16#2E;	//.
    WebPayload[152] := ASCII[1];	//1
    WebPayload[153] := 16#0D;	//<cr>
    WebPayload[154] := 16#0A;	//<nl>
    //Connection:<space>keep-alive<cr><nl>
    WebPayload[155] := 16#43;	//C
    WebPayload[156] := 16#6F;		//o
    WebPayload[157] := 16#6E;	//n
    WebPayload[158] := 16#6E;	//n
    WebPayload[159] := 16#65;	//e
    WebPayload[160] := 16#63;	//c
    WebPayload[161] := 16#74;	//t
    WebPayload[162] := 16#69;	//i
    WebPayload[163] := 16#6F;		//o
    WebPayload[164] := 16#6E;	//n
    WebPayload[165] := 16#3A;	//:
    WebPayload[166] := 16#20;	//<space>
    WebPayload[167] := 16#6B;	//k
    WebPayload[168] := 16#65;	//e
    WebPayload[169] := 16#65;	//e
    WebPayload[170] := 16#70;	//p
    WebPayload[171] := 16#2D;	//-
    WebPayload[172] := 16#61;	//a
    WebPayload[173] := 16#6C;	//l
    WebPayload[174] := 16#69;	//i
    WebPayload[175] := 16#76;	//v
    WebPayload[176] := 16#65;	//e
    WebPayload[177] := 16#0D;	//<cr>
    WebPayload[178] := 16#0A;	//<nl>
    //Content-Length:<space>0<cr><nl><cr><nl>';
    WebPayload[179] := 16#43;	//C
    WebPayload[180] := 16#6F;		//o
    WebPayload[181] := 16#6E;	//n
    WebPayload[182] := 16#74;	//t
    WebPayload[183] := 16#65;	//e
    WebPayload[184] := 16#6E;	//n
    WebPayload[185] := 16#74;	//t
    WebPayload[186] := 16#2D;	//-
    WebPayload[187] := 16#4C;	//L
    WebPayload[188] := 16#65;	//e
    WebPayload[189] := 16#6E;	//n
    WebPayload[190] := 16#67;	//g
    WebPayload[191] := 16#74;	//t
    WebPayload[192] := 16#68;	//h
    WebPayload[193] := 16#3A;	//:
    WebPayload[194] := 16#20;	//<space>
    WebPayload[195] := ASCII[0];	//0
    WebPayload[196] := 16#0D;	//<cr>
    WebPayload[197] := 16#0A;	//<nl>
    WebPayload[198] := 16#0D;	//<cr>
    WebPayload[199] := 16#0A;	//<nl>
    
    //Data_Start := DWORD_TO_STRING(DWORD#218762506); //0D0A0D0A = 218762506
    Data_Start := '$R$L$R$L';
    Manual_Init := 1;
END_IF;
(* Rung 1: Filter analog signals to remove noise *)
IF AGVhasHandheld THEN
    //Exponential filters, alpha is the percentage of new measurement with respect to average
    //alpha is between 0 and 100
    RM_FR1Avg := (alpha*RM_FR1 + (100 - alpha)*RM_FR1Avg)/100;
    RM_LR1Avg := (alpha*RM_LR1 + (100 - alpha)*RM_LR1Avg)/100;
    RM_CenterAvg := (alpha*RM_Center + (100 - alpha)*RM_CenterAvg)/100;
END_IF;
(* Rung 2: Remote control presence check *)
IF AGVhasHandheld THEN
    // Checks if remote is OK
    IF RM_CenterAvg < (CenterCounts*0.8) OR RM_CenterAvg > (CenterCounts*1.2) THEN
    	Remote_Present := FALSE; //Too low center voltage from joystick, remote not connected?
    	HMI_Input10 := FALSE;
    ELSE
    	Remote_Present := TRUE;
    END_IF;
END_IF;

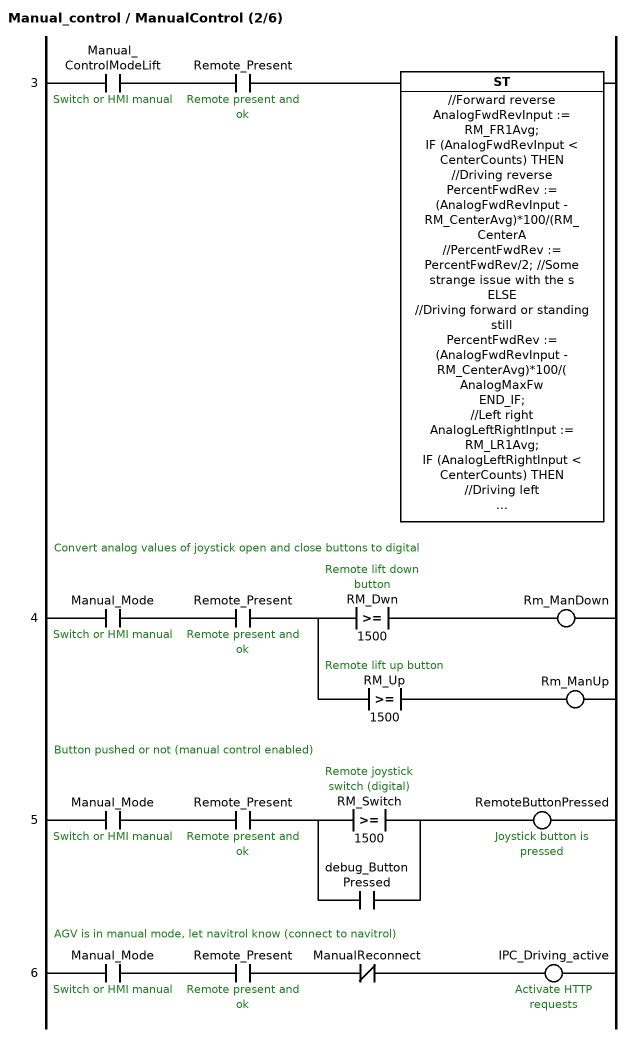
(* Rung 3 *)
IF Manual_ControlModeLift AND Remote_Present THEN
    //Forward reverse
    AnalogFwdRevInput := RM_FR1Avg;
    IF (AnalogFwdRevInput < CenterCounts) THEN
    	 //Driving reverse
    	 PercentFwdRev := (AnalogFwdRevInput - RM_CenterAvg)*100/(RM_CenterAvg - AnalogMaxRevCounts);
    	 //PercentFwdRev := PercentFwdRev/2; //Some strange issue with the schwarzmullers
    ELSE
    	//Driving forward or standing still
    	PercentFwdRev := (AnalogFwdRevInput - RM_CenterAvg)*100/(AnalogMaxFwdCounts - RM_CenterAvg);
    END_IF;
    
    //Left right
    AnalogLeftRightInput := RM_LR1Avg;
    IF (AnalogLeftRightInput < CenterCounts) THEN
    	//Driving left
    	PercentLeftRight:= (AnalogLeftRightInput - RM_CenterAvg)*100/(AnalogMaxRightCounts - RM_CenterAvg);
    ELSE
    	//Driving right or standing still
    	PercentLeftRight := (AnalogLeftRightInput - RM_CenterAvg)*100/(RM_CenterAvg - AnalogMaxLeftCounts);
    END_IF;
END_IF;
(* Rung 4: Convert analog values of joystick open and close buttons to digital *)
Rm_ManDown := Manual_Mode AND Remote_Present AND (RM_Dwn >= 1500);
Rm_ManUp := Manual_Mode AND Remote_Present AND (RM_Up >= 1500);
(* Rung 5: Button pushed or not (manual control enabled) *)
RemoteButtonPressed := Manual_Mode AND Remote_Present AND ((RM_Switch >= 1500) OR debug_ButtonPressed);
(* Rung 6: AGV is in manual mode, let navitrol know (connect to navitrol) *)
IPC_Driving_active := Manual_Mode AND Remote_Present AND NOT ManualReconnect;

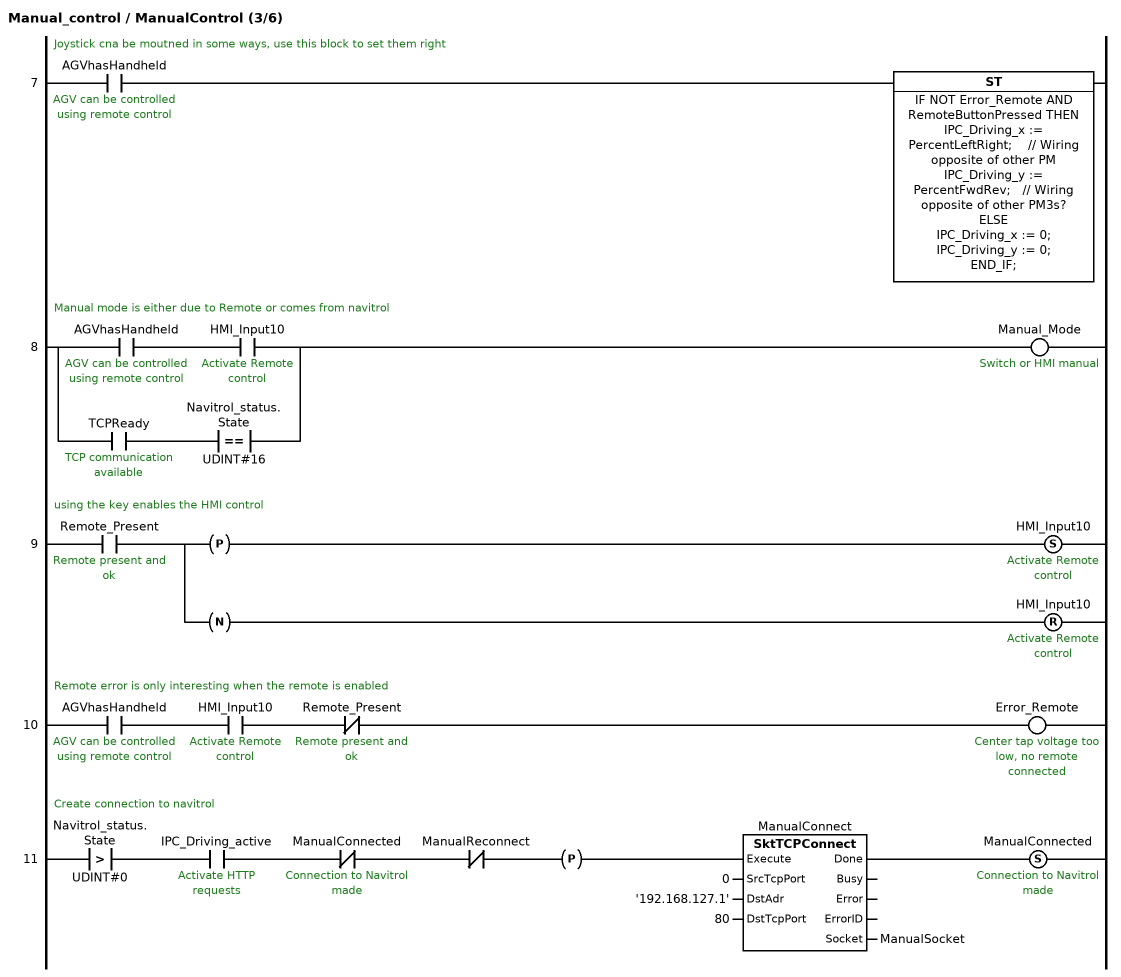
(* Rung 7: Joystick cna be moutned in some ways, use this block to set them right *)
IF AGVhasHandheld THEN
    IF NOT Error_Remote AND RemoteButtonPressed THEN
    	IPC_Driving_x := PercentLeftRight;		// Wiring opposite of other PM3s?
    	IPC_Driving_y := PercentFwdRev;		// Wiring opposite of other PM3s?
    ELSE
    	IPC_Driving_x := 0;
    	IPC_Driving_y := 0;
    END_IF;
END_IF;
(* Rung 8: Manual mode is either due to Remote or comes from navitrol *)
Manual_Mode := (AGVhasHandheld AND HMI_Input10) OR (TCPReady AND (Navitrol_status.State = UDINT#16));
(* Rung 9: using the key enables the HMI control *)
_e1(CLK := Remote_Present);
IF _e1.Q THEN HMI_Input10 := TRUE; END_IF;
_e2(CLK := Remote_Present);
IF _e2.Q THEN HMI_Input10 := FALSE; END_IF;
(* Rung 10: Remote error is only interesting when the remote is enabled *)
Error_Remote := AGVhasHandheld AND HMI_Input10 AND NOT Remote_Present;
(* Rung 11: Create connection to navitrol *)
_e3(CLK := (Navitrol_status.State > UDINT#0) AND IPC_Driving_active AND NOT ManualConnected AND NOT ManualReconnect);
ManualConnect(Execute := _e3.Q, SrcTcpPort := 0, DstAdr := '192.168.127.1', DstTcpPort := 80, Socket => ManualSocket);
IF ManualConnect.Done THEN ManualConnected := TRUE; END_IF;

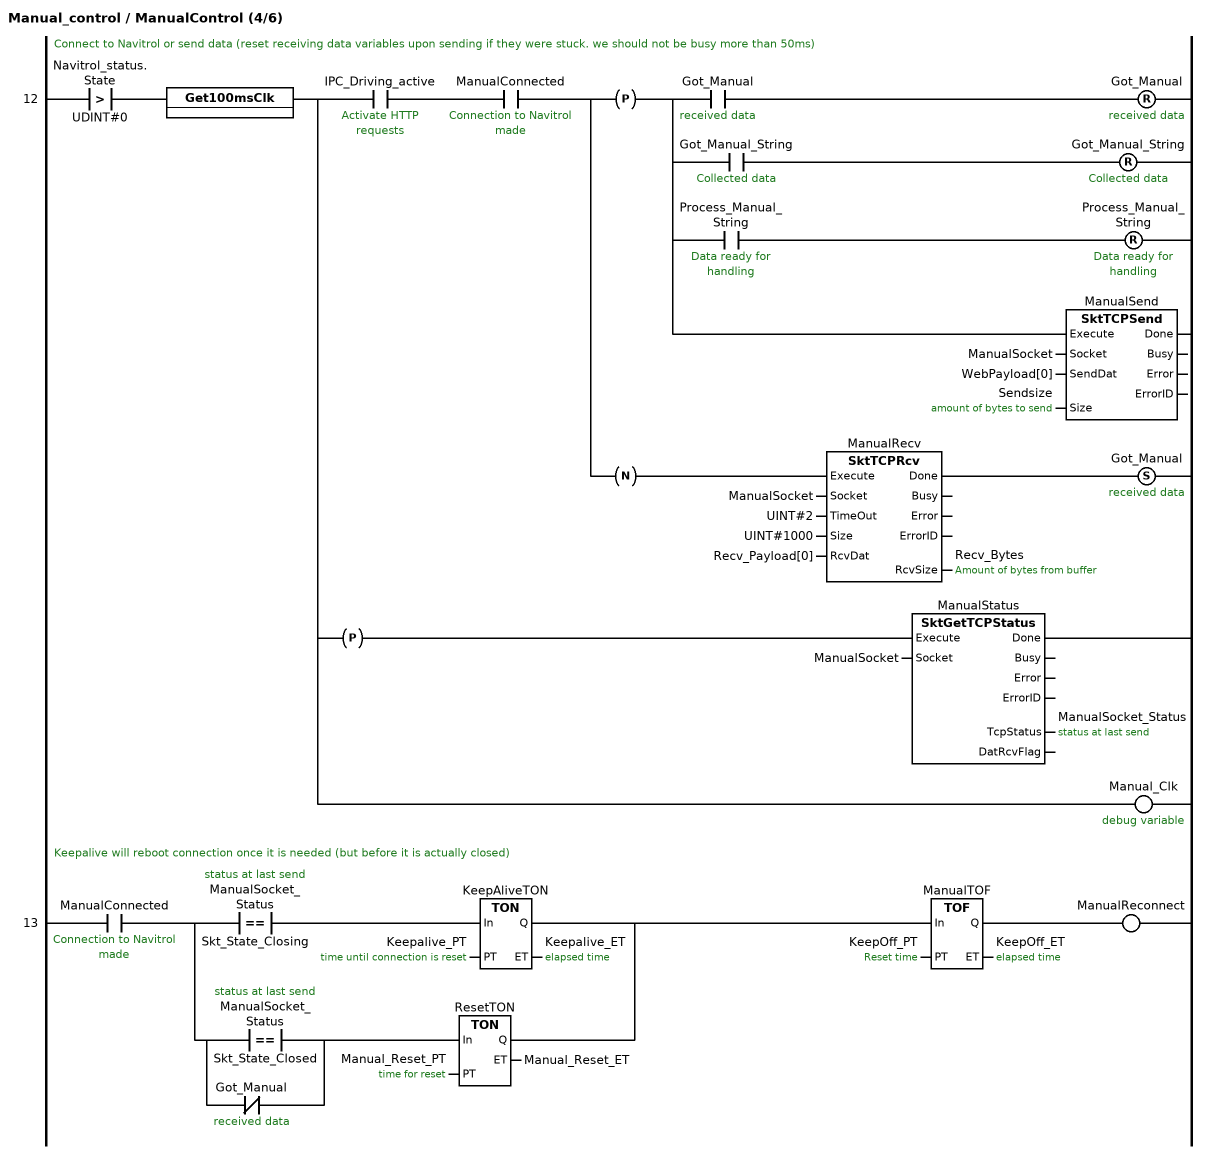
(* Rung 12: Connect to Navitrol or send data (reset receiving data variables upon sending if they were stuck. we should not be busy more than 50ms) *)
_p4 := (Navitrol_status.State > UDINT#0) AND Get100msClk();
_e5(CLK := _p4 AND IPC_Driving_active AND ManualConnected);
IF _e5.Q AND Got_Manual THEN Got_Manual := FALSE; END_IF;
IF _e5.Q AND Got_Manual_String THEN Got_Manual_String := FALSE; END_IF;
IF _e5.Q AND Process_Manual_String THEN Process_Manual_String := FALSE; END_IF;
ManualSend(Execute := _e5.Q, Socket := ManualSocket, SendDat := WebPayload[0], Size := Sendsize);
_e6(CLK := _p4 AND IPC_Driving_active AND ManualConnected);
ManualRecv(Execute := _e6.Q, Socket := ManualSocket, TimeOut := UINT#2, Size := UINT#1000, RcvDat := Recv_Payload[0], RcvSize => Recv_Bytes);
IF ManualRecv.Done THEN Got_Manual := TRUE; END_IF;
_e7(CLK := _p4);
ManualStatus(Execute := _e7.Q, Socket := ManualSocket, TcpStatus => ManualSocket_Status);
Manual_Clk := _p4;
(* Rung 13: Keepalive will reboot connection once it is needed (but before it is actually closed) *)
KeepAliveTON(In := ManualConnected AND (ManualSocket_Status = Skt_State_Closing), PT := Keepalive_PT, ET => Keepalive_ET);
ResetTON(In := ManualConnected AND ((ManualSocket_Status = Skt_State_Closed) OR NOT Got_Manual), PT := Manual_Reset_PT, ET => Manual_Reset_ET);
ManualTOF(In := KeepAliveTON.Q OR ResetTON.Q, PT := KeepOff_PT, ET => KeepOff_ET);
ManualReconnect := ManualTOF.Q;

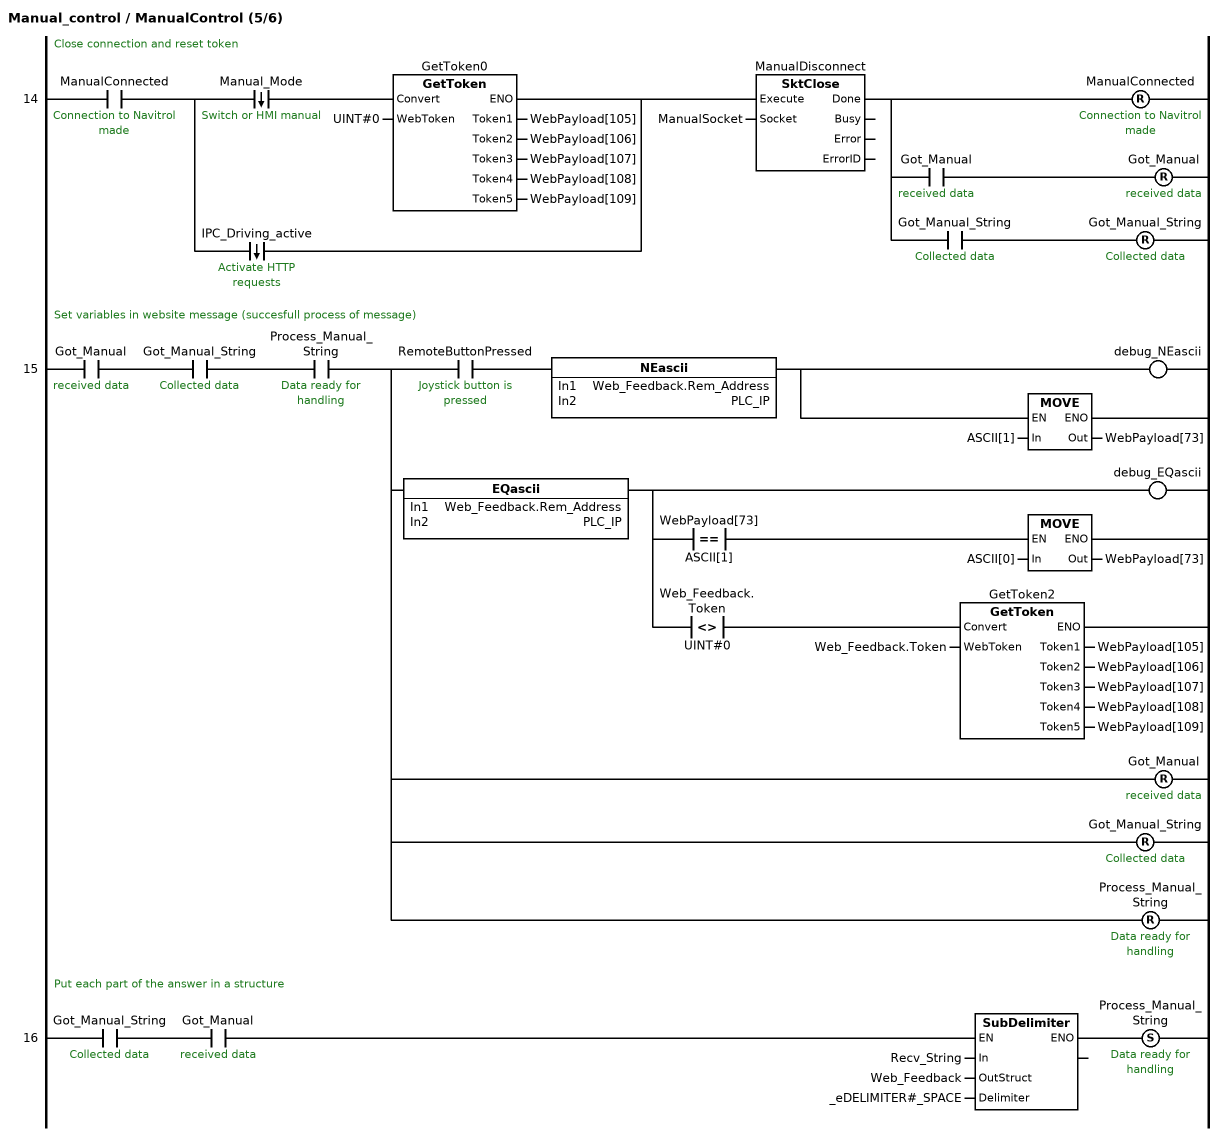
(* Rung 14: Close connection and reset token *)
_e8(CLK := Manual_Mode);
GetToken0(Convert := ManualConnected AND _e8.Q, WebToken := UINT#0, Token1 => WebPayload[105], Token2 => WebPayload[106], Token3 => WebPayload[107], Token4 => WebPayload[108], Token5 => WebPayload[109]);
_e9(CLK := IPC_Driving_active);
ManualDisconnect(Execute := GetToken0.ENO OR (ManualConnected AND _e9.Q), Socket := ManualSocket);
IF ManualDisconnect.Done THEN ManualConnected := FALSE; END_IF;
IF ManualDisconnect.Done AND Got_Manual THEN Got_Manual := FALSE; END_IF;
IF ManualDisconnect.Done AND Got_Manual_String THEN Got_Manual_String := FALSE; END_IF;
(* Rung 15: Set variables in website message (succesfull process of message) *)
_p10 := Got_Manual AND Got_Manual_String AND Process_Manual_String;
_p11 := _p10 AND RemoteButtonPressed AND NEascii(Web_Feedback.Rem_Address, PLC_IP);
debug_NEascii := _p11;
IF _p11 THEN WebPayload[73] := ASCII[1]; END_IF;
_p12 := _p10 AND EQascii(Web_Feedback.Rem_Address, PLC_IP);
debug_EQascii := _p12;
IF _p12 AND (WebPayload[73] = ASCII[1]) THEN WebPayload[73] := ASCII[0]; END_IF;
GetToken2(Convert := _p12 AND (Web_Feedback.Token <> UINT#0), WebToken := Web_Feedback.Token, Token1 => WebPayload[105], Token2 => WebPayload[106], Token3 => WebPayload[107], Token4 => WebPayload[108], Token5 => WebPayload[109]);
IF _p10 THEN
    Got_Manual := FALSE;
    Got_Manual_String := FALSE;
    Process_Manual_String := FALSE;
END_IF;
(* Rung 16: Put each part of the answer in a structure *)
IF Got_Manual_String AND Got_Manual THEN
    SubDelimiter(In := Recv_String, OutStruct := Web_Feedback, Delimiter := _eDELIMITER#_SPACE);
    Process_Manual_String := TRUE;
END_IF;

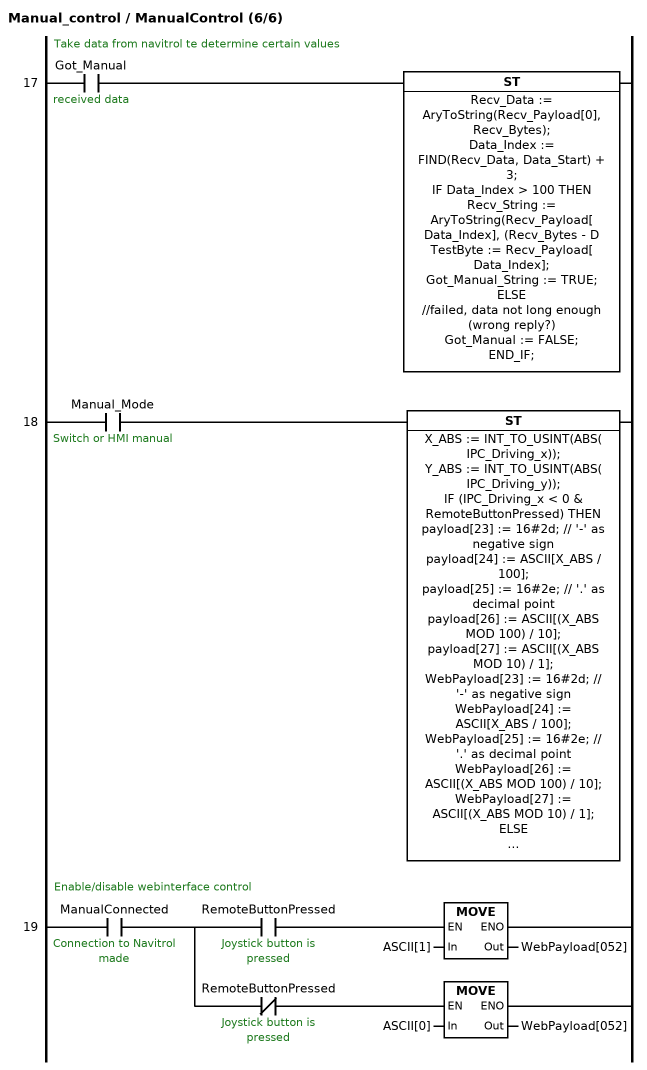
(* Rung 17: Take data from navitrol te determine certain values *)
_p13 := Got_Manual;
IF _p13 THEN
    Recv_Data := AryToString(Recv_Payload[0], Recv_Bytes);
    Data_Index := FIND(Recv_Data, Data_Start) + 3;
    IF Data_Index > 100 THEN
    	Recv_String := AryToString(Recv_Payload[Data_Index], (Recv_Bytes - Data_Index));
    	TestByte := Recv_Payload[Data_Index];
    	Got_Manual_String := TRUE;
    ELSE
    	//failed, data not long enough (wrong reply?)
    	Got_Manual := FALSE;
    END_IF;
END_IF;
(* Rung 18 *)
IF Manual_Mode THEN
    X_ABS := INT_TO_USINT(ABS(IPC_Driving_x));
    Y_ABS := INT_TO_USINT(ABS(IPC_Driving_y));
    IF (IPC_Driving_x < 0 & RemoteButtonPressed) THEN
    	payload[23] := 16#2d; // '-' as negative sign
    	payload[24] := ASCII[X_ABS / 100];
    	payload[25] := 16#2e; // '.' as decimal point
    	payload[26] := ASCII[(X_ABS MOD 100) / 10];
    	payload[27] := ASCII[(X_ABS MOD 10) / 1];
    	
    	WebPayload[23] := 16#2d; // '-' as negative sign
    	WebPayload[24] := ASCII[X_ABS / 100];
    	WebPayload[25] := 16#2e; // '.' as decimal point
    	WebPayload[26] := ASCII[(X_ABS MOD 100) / 10];
    	WebPayload[27] := ASCII[(X_ABS MOD 10) / 1];
    ELSE
    	payload[23] := ASCII[X_ABS / 100];
    	payload[24] := 16#2e; // '.' as decimal point
    	payload[25] := ASCII[(X_ABS MOD 100) / 10];
    	payload[26] := ASCII[(X_ABS MOD 10) / 1];
    	payload[27] := ASCII[0]; // trailing zero
    	
    	WebPayload[23] := ASCII[X_ABS / 100];
    	WebPayload[24] := 16#2e; // '.' as decimal point
    	WebPayload[25] := ASCII[(X_ABS MOD 100) / 10];
    	WebPayload[26] := ASCII[(X_ABS MOD 10) / 1];
    	WebPayload[27] := ASCII[0]; // trailing zero
    END_IF;
    IF (IPC_Driving_y < 0 & RemoteButtonPressed) THEN
    	payload[31] := 16#2d; // '-' as negative sign
    	payload[32] := ASCII[Y_ABS / 100];
    	payload[33] := 16#2e; // '.' as decimal point
    	payload[34] := ASCII[(Y_ABS MOD 100) / 10];
    	payload[35] := ASCII[(Y_ABS MOD 10) / 1];
    	
    	WebPayload[31] := 16#2d; // '-' as negative sign
    	WebPayload[32] := ASCII[Y_ABS / 100];
    	WebPayload[33] := 16#2e; // '.' as decimal point
    	WebPayload[34] := ASCII[(Y_ABS MOD 100) / 10];
    	WebPayload[35] := ASCII[(Y_ABS MOD 10) / 1];
    ELSE
    	payload[31] := ASCII[Y_ABS / 100];
    	payload[32] := 16#2e; // '.' as decimal point
    	payload[33] := ASCII[(Y_ABS MOD 100) / 10];
    	payload[34] := ASCII[(Y_ABS MOD 10) / 1];
    	payload[35] := ASCII[0]; // trailing zero
    	
    	WebPayload[31] := ASCII[Y_ABS / 100];
    	WebPayload[32] := 16#2e; // '.' as decimal point
    	WebPayload[33] := ASCII[(Y_ABS MOD 100) / 10];
    	WebPayload[34] := ASCII[(Y_ABS MOD 10) / 1];
    	WebPayload[35] := ASCII[0]; // trailing zero
    END_IF;
END_IF;
(* Rung 19: Enable/disable webinterface control *)
IF ManualConnected AND RemoteButtonPressed THEN WebPayload[052] := ASCII[1]; END_IF;
IF ManualConnected AND NOT RemoteButtonPressed THEN WebPayload[052] := ASCII[0]; END_IF;
END_PROGRAM

PROGRAM Navitrol
VAR
    PLC_Manual : PLC_Navitrol_Manual_struct;
    PLC_err : PLC_Err_sec_struct;  (* PLC error heading struct *)
    PLC_Navitrol_Joystick : PLC_Navitrol_Joystick_struct;
    PLC_Navitrol_Drivecontrol : PLC_Navitrol_DriveControl_struct;
    PLC_Navitrol_Battery : Navitrol_Status_Battery_struct;
    CoError : BOOL;  (* Socket open error *)
    CoOpen : BOOL;  (* open socket *)
    CoDone : BOOL;  (* TCP socket opened *)
    CoClose : BOOL;  (* close socket *)
    ClDone : BOOL;  (* Close complete *)
    ClBusy : BOOL;  (* Closing socket *)
    StDone : BOOL;  (* TCP status updated *)
    CoBusy : BOOL;  (* Socket being opened *)
    CoErrorID : WORD;  (* Error ID *)
    TcpSocket : _sSOCKET;  (* Navitrol socket *)
    RcvFlag : BOOL;  (* Data in RX buffer *)
    RxResetElapsedTime : TIME;  (* elapsed time *)
    ClError : BOOL;  (* Closing encountered error *)
    ClErrorID : WORD;  (* Error ID *)
    StBusy : BOOL;  (* Update in progress *)
    StError : BOOL;  (* Update encountered error *)
    StErrorID : WORD;  (* Error ID *)
    TCPStatus : _eCONNECTION_STATE;  (* Socket status *)
    Connect_Inst : SktTCPConnect;
    Close_Inst : SktClose;
    Status_Inst : SktGetTCPStatus;
    StatusDelay_TON : TON;
    StatusDelay_TON_Time : TIME;  (* Status timer *)
    PauseMessageID : UINT;  (* Message ID *)
    ResumeMessageID : UINT;  (* Message ID *)
    TxSupervisorStatus : SendSupervisorStatus;
    StatusBusy : BOOL;  (* Status is being send *)
    StatusDone : BOOL;  (* Transmission completed *)
    SpeedArrayBusy : BOOL;  (* Transmission in progress *)
    Zeroseconds : TIME := 0s;  (* 0s *)
    RxResetTimeSetpoint : TIME := 5s;  (* Rx timeout *)
    RxResetTimer : TON;
    DataIn : ARRAY[0..1023] OF BYTE;  (* Raw bytes; [0] Full raw data *)
    RcvBusy : BOOL;  (* Rx in progress *)
    RcvError : BOOL;  (* Error during receive action *)
    RcvErrorID : WORD;  (* Error ID *)
    RcvSize : UINT;  (* Bytes actually read *)
    Recv_Inst : SktTCPRcv;
    Order : _eBYTE_ORDER := _LOW_HIGH;  (* byte order *)
    RecvProtocol : UINT;  (* Received protocol version *)
    RecvID : UINT;  (* Received message ID *)
    RecvLength : UDINT;  (* Received frame size *)
    RecvLength_UINT : UINT;  (* Received frame size *)
    CheckData : BOOL;  (* Checking received data before processing *)
    DataOk : BOOL;  (* Data seems ok *)
    DataNok : BOOL;  (* Data invalid *)
    RxNavitrolStatus : ReceiveNavitrolStatus;
    RxStatusBusy : BOOL;  (* Busy with data *)
    RxResetData : TON;
    TimeoutRx : TIME;  (* Time RX may remain stuck *)
    RxStuckTime : TIME;  (* Time RX does not change *)
    KeepRxClosed_TP : TP;
    KeepRxClosed_PT : TIME := 1s;  (* Time RX should remain offline *)
    KeepRxClosed_ET : TIME;  (* elapsed time *)
    RxSendTargetDetectionUpdate : ReceiveNavitrol4101;
    Navitrol_TargetUpdate : Navitrol_TargetDetUpdate_struct;  (* Target calculation complete *)
    RxTargetDetectionStatus : ReceiveNavitrol4105;
    Navitrol_TargetDetection : Navitrol_TargetDetStatus_struct;  (* Navitrol target found message *)
    PalletDetectionSettings : Navitrol_SetTargetDetectionControlModeLift_struct;  (* Settings for navitrol pallet detetction *)
    TxMessage3006 : SendPauseDrive;
    TxMessage3007 : SendResumeDrive;
    TxMessage3008 : SendAbortDrive;
    TxMessage3028 : SendSetSpeedArray;
    RequestNavitrolLog : BOOL;  (* Ask navitrol to make a log *)
    TxMessage1007 : SendSaveLog;
    AbortNavitrolDrive : BOOL;  (* Abort navitrol drive with data *)
    TxMessage3032 : SendSetTargetDetectionMode;
    TxMessage3023 : SendSetSpeedLimit;
    Navitrol_ErrorCount : UDINT;  (* Amount of active navitrol errors *)
    Navitrol_ErrorList : ARRAY[0..9] OF UDINT;  (* Array of max 10 errors active in navitrol *)
    ReceiveNavitrolErrorList : ReceiveNavitrol201;
    Navitrol_PauseResult : UDINT;  (* 0=ok, 1=bad input, 2=wrong state *)
    Navitrol_Savelog_Result : UDINT;  (* 0=fail, else number of log *)
    Navitrol_ResumeID : UDINT;  (* Resuming to symbolic point ID *)
    Navitrol_ResumeResult : UDINT;  (* 0=ok, 1=bad input, 2=wrong state *)
    Navitrol_AbortResult : UDINT;  (* 0=ok, 1=bad input, 2=wrong state *)
    Navitrol_SpeedSet : UINT;  (* 0=released, 1=set *)
    Navitrol_SpeedLimit : REAL;  (* Max speed or max value (released) *)
    Navitrol_ArraySet : UINT;  (* 0=array released, 1=array set *)
    Navitrol_DriveReady : UDINT;  (* 0=Ok, 1=Fail *)
    TxMessage3033 : SendAbortWithData;
    DriveDone : BOOL;  (* 1: drive completed *)
    TxMessage3038 : SendRequestDriveReady;
    TestData : ARRAY[0..1023] OF BYTE;  (* compare data *)
    ReDone : BOOL;  (* Raw data received *)
    TxMessage3014 : SendRequestProductionStatus;
    TxMessage3009 : SendAbortDrive;
    debug_ReqError : BOOL;
    TxMessage3040 : SendAckFatal;
END_VAR
VAR_EXTERNAL
    AGVusesActuator : BOOL;
    PLC_status : PLC_Status_Struct;
    MessageLength : UDINT;
    NrOfSections : UINT;
    PLC_act : PLC_Act_Sec_Struct;
    Navitrol_ManualSection_Enabled : BOOL;
    Navitrol_ErrorSection_Enabled : BOOL;
    PLC_Error_Array : array[0..4] of PLC_Error_struct;
    Navitrol_InputSection_Enabled : BOOL;
    PLC_Navitrol_input : Navitrol_Status_inputs_struct;
    NumBytes : UINT;
    NumInts : UINT;
    NumFloats : UINT;
    Navitrol_LaserSection_Enabled : BOOL;
    PLC_Navitrol_laserscanners : PLC_Navitrol_Status_laserscanner_struct;
    Navitrol_RemoteControlSection_Enabled : BOOL;
    Navitrol_Drivecontrol_Enabled : BOOL;
    Navitrol_PLC_Battery_Enabled : BOOL;
    AGV_Init : UINT;
    TCPReady : BOOL;
    Navitrol_RX_Port : UINT;
    Navitrol_IP : STRING[256];
    Navitrol_TX_Port : UINT;
    Update_Navitrol : BOOL;
    SpeedArray : UINT;
    PLC_Warn_Array : array[0..4] of PLC_Warn_struct;
    Navitrol_status : Navitrol_Status_Struct;
    Navitrol_gen : Navitrol_Status_General_Sec_Struct;
    Navitrol_Tag : Navitrol_Status_TagV4_sec_struct;
    Navitrol_FromTo : Navitrol_Status_FromTo_Sec_struct;
    Navitrol_act : Navitrol_Status_Act_Sec_Struct;
    Navitrol_Steer : Navitrol_Status_Steering_Sec_Struct;
    NavitrolPause : BOOL;
    NavitrolResume : BOOL;
    Navitrol_Battery : Navitrol_Status_Battery_struct;  (* Battery status from navitrol *)
    SendTargetDetectionSettings : BOOL;  (* send message 3202 to navitrol *)
    NavitrolAbort : BOOL;  (* Request navitrol to abort drive *)
    Navitrol_DistanceInfo : Navitrol_Status_DistanceToTarget_sec_struct;  (* Driveorder information *)
    SetNavitrolSpeedLimit : BOOL;  (* Send true to use speed limiter *)
    SpeedLimit : REAL;  (* Max speed in m/s for limiter message *)
    Navitrol_SpeedUpdate : BOOL;
    NavitrolSpeedLimit : BOOL;
    NavitrolArrayLimit : BOOL;
    Navitrol_DriveInfo : Navitrol_Status_DriveorderInfo_sec_struct;  (* Driveinfo section *)
    Manual_Navitrol : BOOL;  (* Navitrol in manual state *)
    RequestDriveReady : BOOL;  (* Target reached *)
    DriveType : UINT;  (* Request ready tpe *)
    Sections : ARRAY[1..10] OF UINT;
    RequestProductionStatus : BOOL;  (* Request the production status data from Navitrol *)
    Navitrol_ProductionStatus : Navitrol_ProductionData_struct;
    Navitrol_ProdDataStatusResult : UINT;  (* 0=not activated, 1=activated *)
    Navitrol_Cust : Navitrol_Status_Custom_sec_struct;  (* Navitrol status, custom attribute *)
    Navitrol_TargetDetectionStatus : Navitrol_TargetDetectionStatus_struct;
    Navitrol_ErrorWithLevel : Navitrol_ErrorWithLevel_Struct;
    todo : BOOL;
    BufferLaneNavitrol_speed_limiter : BOOL;
END_VAR
VAR
    _p1 : BOOL;
    _p2 : BOOL;
    _e3 : R_TRIG;
    _e4 : R_TRIG;
    _p5 : BOOL;
    _p6 : BOOL;
    _p7 : BOOL;
    _p8 : BOOL;
    _p9 : BOOL;
    _p10 : BOOL;
    _p11 : BOOL;
    _p12 : BOOL;
    _p13 : BOOL;
    _p14 : BOOL;
    _p15 : BOOL;
    _p16 : BOOL;
    _p17 : BOOL;
    _p18 : BOOL;
    _p19 : BOOL;
    _p20 : BOOL;
    _p21 : BOOL;
END_VAR

(* Section Core: ladder, written here as Structured Text *)

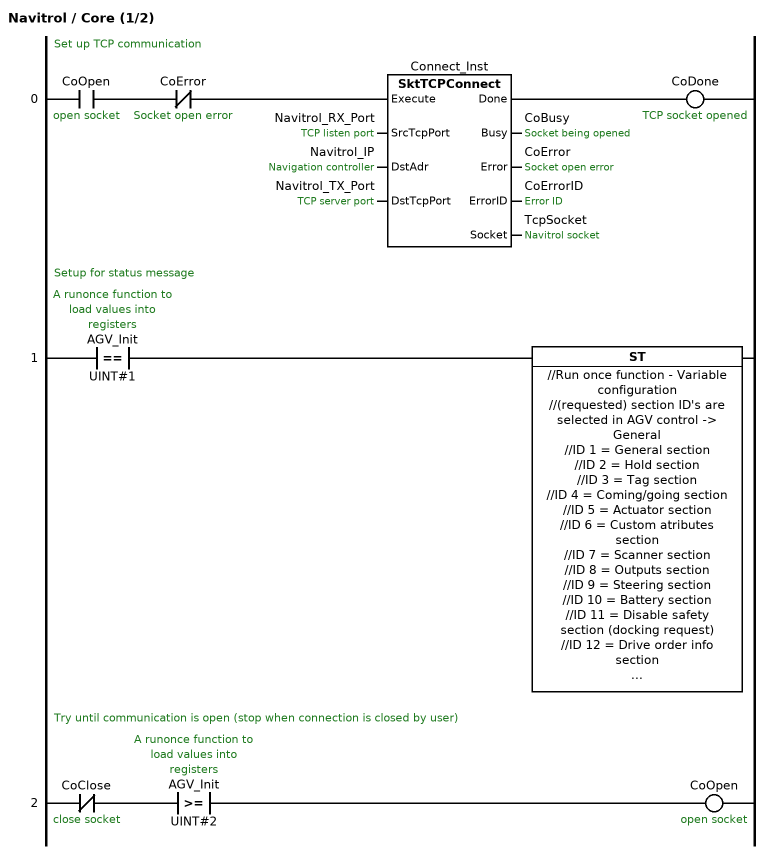
(* Rung 0: Set up TCP communication *)
_p1 := CoOpen AND NOT CoError;
Connect_Inst(Execute := _p1, SrcTcpPort := Navitrol_RX_Port, DstAdr := Navitrol_IP, DstTcpPort := Navitrol_TX_Port, Busy => CoBusy, Error => CoError, ErrorID => CoErrorID, Socket => TcpSocket);
CoDone := Connect_Inst.Done;
(* Rung 1: Setup for status message *)
IF AGV_Init = UINT#1 THEN
    //Run once function - Variable configuration
    
    //(requested) section ID's are selected in AGV control -> General
    //ID 1 = General section
    //ID 2 = Hold section
    //ID 3 = Tag section
    //ID 4 = Coming/going section
    //ID 5 = Actuator section
    //ID 6 = Custom atributes section
    //ID 7 = Scanner section
    //ID 8 = Outputs section
    //ID 9 = Steering section
    //ID 10 = Battery section
    //ID 11 = Disable safety section (docking request)
    //ID 12 = Drive order info section
    //ID 13 = Distance to target section
    
    PLC_status.Prot_Ver := 4;
    PLC_status.Message_ID := 3002;
    MessageLength := 14;		//base message length is 14 bytes
    
    //Amount of requested sections is added to message length
    MessageLength := MessageLength + (2*NrOfSections);
    
    //PLC Actuator variables set
    IF (AGVusesActuator) THEN
    	//the rest of actuator section variables are set in AGV_Control -> general
    	MessageLength := MessageLength + PLC_act.Section_Length;
    	PLC_act.B_Inp.Load_Sensor_In_Use := TRUE;
    END_IF;
    
    //Manual section (keyboard control)
    IF (Navitrol_ManualSection_Enabled) THEN
    	PLC_Manual.Section_ID := 2;
    	PLC_Manual.Section_length := 20;	//fixed message length
    	PLC_Manual.Auto_Manual := 0;		//start disabled
    END_IF;
    
    //Error section
    IF (Navitrol_ErrorSection_Enabled) THEN
    	//test error and warning message
    	PLC_err.Section_ID := 3;
    	
    	//message length is dependand on active errors and warnings. Only the minimal is added at all times and more is added at TX
    	MessageLength := MessageLength + 10;
    END_IF;
    
    //inputs section
    IF (Navitrol_InputSection_Enabled) THEN
    	PLC_Navitrol_input.Section_ID := 4;
    	//amount of bytes, int and floats (reals) are set in AGV_Control -> general
    	PLC_Navitrol_input.Section_Length := 12 + NumBytes + (4*NumInts) + (4*NumFloats);
    	PLC_Navitrol_input.NumberOfBytes := NumBytes;
    	PLC_Navitrol_input.NumberOfInts := NumInts;
    	PLC_Navitrol_input.NumberOfFloats := NumFloats;
    	MessageLength := MessageLength + PLC_Navitrol_input.Section_Length;
    END_IF;
    
    //safety scanner section
    IF (Navitrol_LaserSection_Enabled) THEN
    	PLC_Navitrol_laserscanners.Section_ID := 5;
    	PLC_Navitrol_laserscanners.Section_Length := 12;
    	MessageLength := MessageLength + PLC_Navitrol_laserscanners.Section_Length;
    END_IF;
    
    //joystick to navitrol section
    IF (Navitrol_RemoteControlSection_Enabled) THEN
    	PLC_Navitrol_Joystick.Section_ID := 6;
    	PLC_Navitrol_Joystick.Section_length := 28;
    	PLC_Navitrol_Joystick.Remote_control2 := 0;	//no lift control (handled by IO)
    	PLC_Navitrol_Joystick.Joystick2_X := 0;
    	PLC_Navitrol_Joystick.Joystick2_Y := 0;
    	PLC_Navitrol_Joystick.Controlmode := 1; //unused for non-omni AGVs
    	//1 = Omni Front wheel steer, 2 = Omni Mid wheel steer, 3 = Omni Rear wheel steer, 4 = Not used
    	//5 = Pivot steer, 6 = Omni Parallel steer, wheeling Fwd, 7 = Omni Parallel steer, wheeling Bwd
    END_IF;
    
    //drive control section (disable certain drive commands)
    IF (Navitrol_Drivecontrol_Enabled) THEN
    	PLC_Navitrol_Drivecontrol.Section_ID := 7;
    	PLC_Navitrol_Drivecontrol.Section_length := 8;
    END_IF;
    
    //battery section (to navitrol)
    IF (Navitrol_PLC_Battery_Enabled) THEN
    	//battery information to navitrol. requires parameter I,extbatt_if_type = 5 in navitrol parameters
    	PLC_Navitrol_Battery.Section_ID := 8;
    	PLC_Navitrol_Battery.Section_length := 30;
    END_IF;
    
    //add final information to structure
    PLC_status.Message_Length := MessageLength;
    PLC_status.Nmbr_Of_Sec := NrOfSections;
    
    //Message IDs
    PauseMessageID := 3006;
    ResumeMessageID := 3007;
    
    //SetTargetDetection
    PalletDetectionSettings.ProtocolVersion := 4;
    PalletDetectionSettings.Message_ID := 3032;
    PalletDetectionSettings.Message_length := 48;
    PalletDetectionSettings.TargetDetectionControlModeLift := 2;	//pallet detection v2
    PalletDetectionSettings.PalletsToDetect := 0;				//all ControlModeLiftls off
    
    //run once procedure completed, ready to open socket
    AGV_Init := AGV_Init +1;
END_IF;
(* Rung 2: Try until communication is open (stop when connection is closed by user) *)
CoOpen := NOT CoClose AND (AGV_Init >= UINT#2);

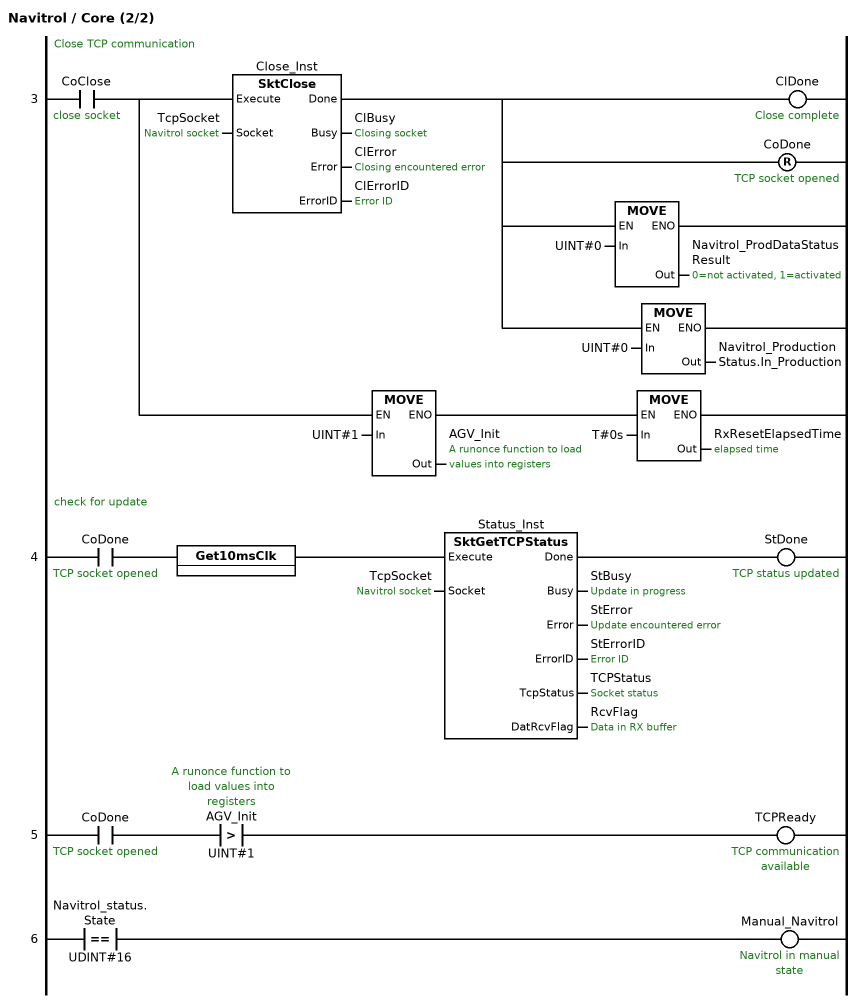
(* Rung 3: Close TCP communication *)
Close_Inst(Execute := CoClose, Socket := TcpSocket, Busy => ClBusy, Error => ClError, ErrorID => ClErrorID);
ClDone := Close_Inst.Done;
IF Close_Inst.Done THEN
    CoDone := FALSE;
    Navitrol_ProdDataStatusResult := UINT#0;
    Navitrol_ProductionStatus.In_Production := UINT#0;
END_IF;
IF CoClose THEN
    AGV_Init := UINT#1;
    RxResetElapsedTime := T#0s;
END_IF;
(* Rung 4: check for update *)
Status_Inst(Execute := CoDone AND Get10msClk(), Socket := TcpSocket, Busy => StBusy, Error => StError, ErrorID => StErrorID, TcpStatus => TCPStatus, DatRcvFlag => RcvFlag);
StDone := Status_Inst.Done;
(* Rung 5 *)
TCPReady := CoDone AND (AGV_Init > UINT#1);
(* Rung 6 *)
Manual_Navitrol := Navitrol_status.State = UDINT#16;

(* Section Tx: ladder, written here as Structured Text *)

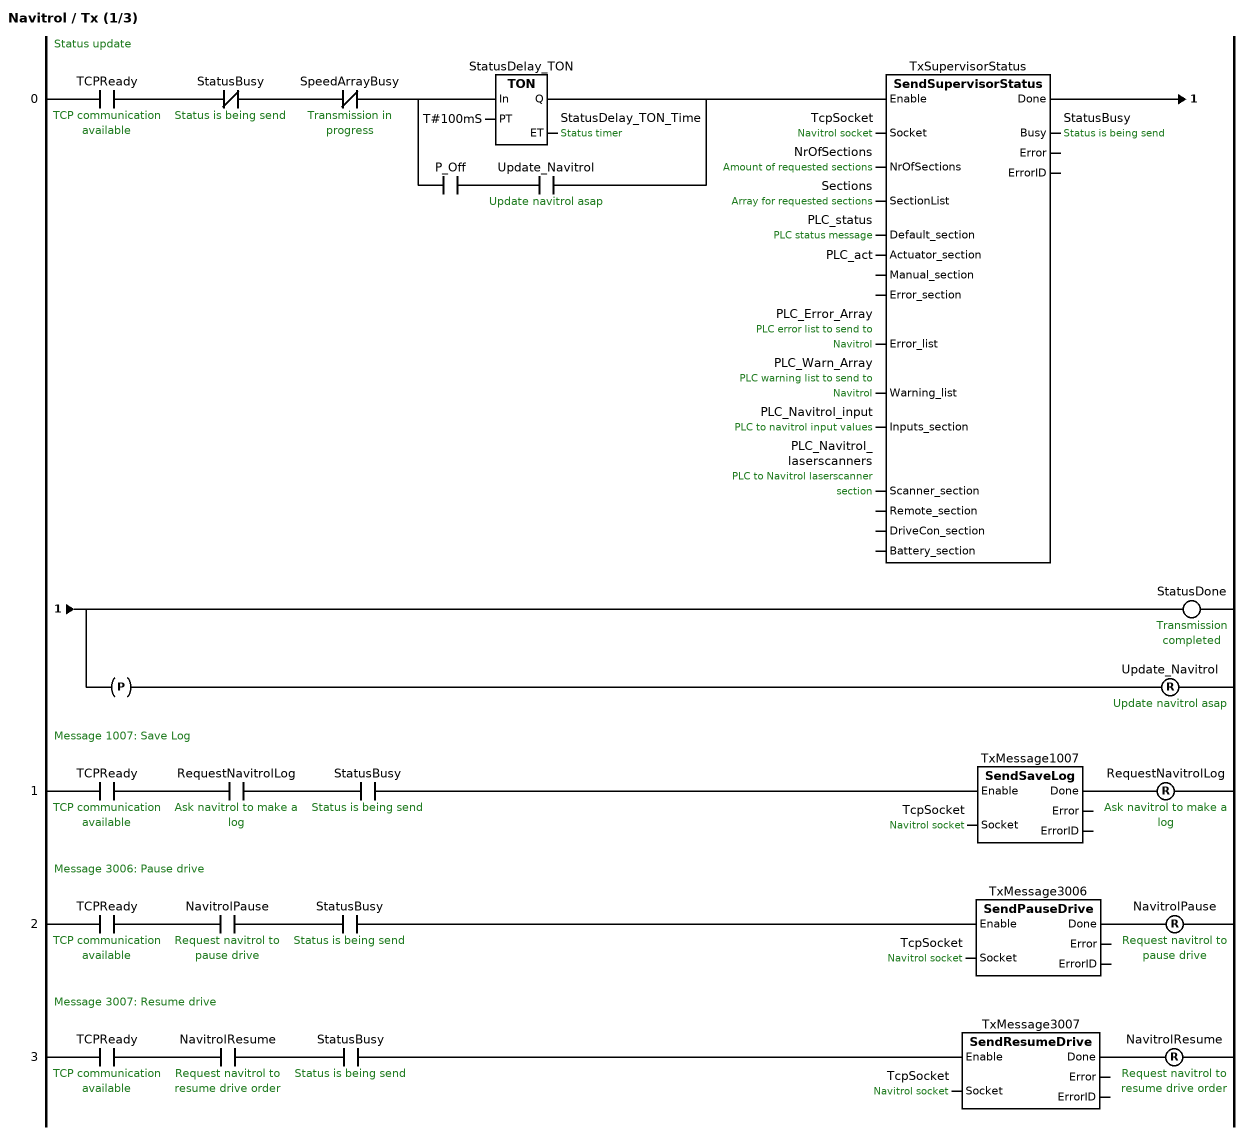
(* Rung 0: Status update *)
_p2 := TCPReady AND NOT StatusBusy AND NOT SpeedArrayBusy;
StatusDelay_TON(In := _p2, PT := T#100mS, ET => StatusDelay_TON_Time);
TxSupervisorStatus(Enable := StatusDelay_TON.Q OR (_p2 AND P_Off AND Update_Navitrol), Socket := TcpSocket, NrOfSections := NrOfSections, SectionList := Sections, Default_section := PLC_status, Actuator_section := PLC_act, Error_list := PLC_Error_Array, Warning_list := PLC_Warn_Array, Inputs_section := PLC_Navitrol_input, Scanner_section := PLC_Navitrol_laserscanners, Busy => StatusBusy);
StatusDone := TxSupervisorStatus.Done;
_e3(CLK := TxSupervisorStatus.Done);
IF _e3.Q THEN Update_Navitrol := FALSE; END_IF;
(* Rung 1: Message 1007: Save Log *)
TxMessage1007(Enable := TCPReady AND RequestNavitrolLog AND StatusBusy, Socket := TcpSocket);
IF TxMessage1007.Done THEN RequestNavitrolLog := FALSE; END_IF;
(* Rung 2: Message 3006: Pause drive *)
TxMessage3006(Enable := TCPReady AND NavitrolPause AND StatusBusy, Socket := TcpSocket);
IF TxMessage3006.Done THEN NavitrolPause := FALSE; END_IF;
(* Rung 3: Message 3007: Resume drive *)
TxMessage3007(Enable := TCPReady AND NavitrolResume AND StatusBusy, Socket := TcpSocket);
IF TxMessage3007.Done THEN NavitrolResume := FALSE; END_IF;

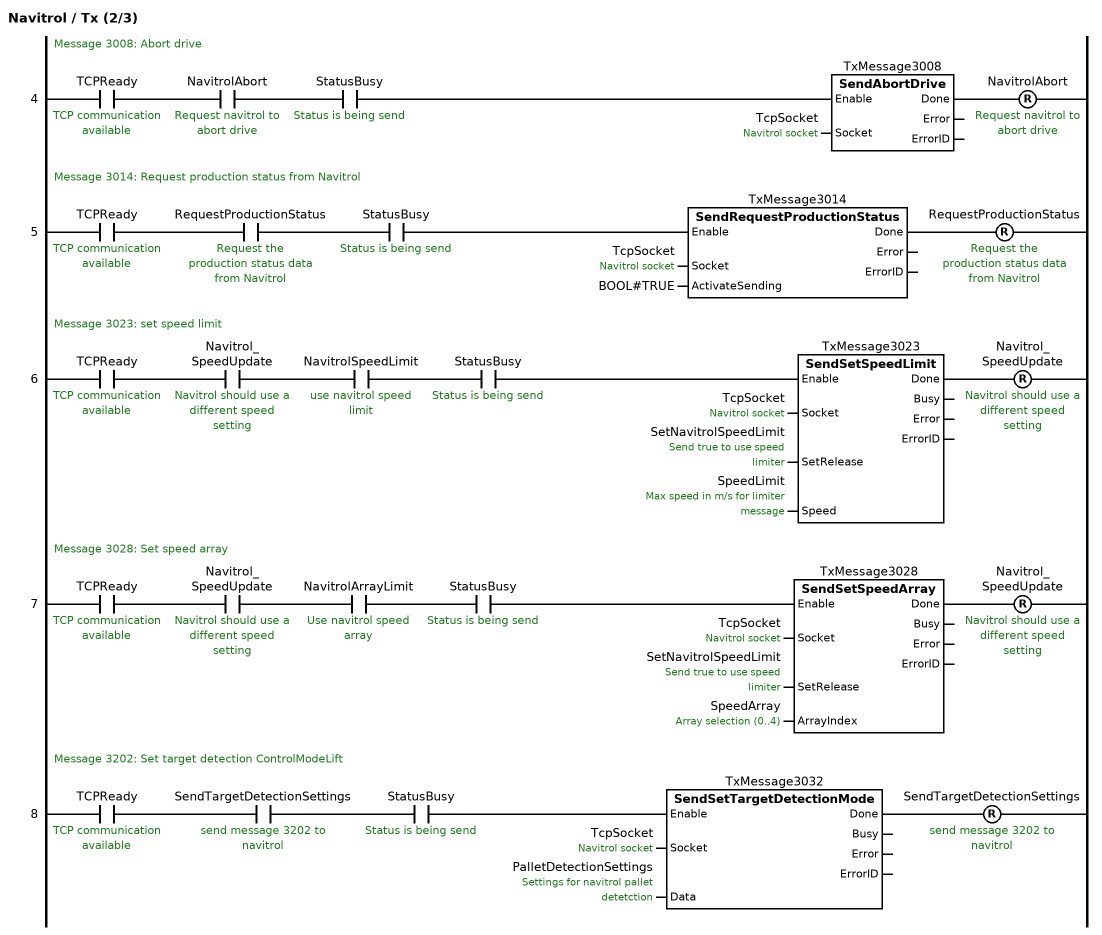
(* Rung 4: Message 3008: Abort drive *)
TxMessage3008(Enable := TCPReady AND NavitrolAbort AND StatusBusy, Socket := TcpSocket);
IF TxMessage3008.Done THEN NavitrolAbort := FALSE; END_IF;
(* Rung 5: Message 3014: Request production status from Navitrol *)
TxMessage3014(Enable := TCPReady AND RequestProductionStatus AND StatusBusy, Socket := TcpSocket, ActivateSending := BOOL#TRUE);
IF TxMessage3014.Done THEN RequestProductionStatus := FALSE; END_IF;
(* Rung 6: Message 3023: set speed limit *)
TxMessage3023(Enable := TCPReady AND Navitrol_SpeedUpdate AND NavitrolSpeedLimit AND StatusBusy, Socket := TcpSocket, SetRelease := SetNavitrolSpeedLimit, Speed := SpeedLimit);
IF TxMessage3023.Done THEN Navitrol_SpeedUpdate := FALSE; END_IF;
(* Rung 7: Message 3028: Set speed array *)
TxMessage3028(Enable := TCPReady AND Navitrol_SpeedUpdate AND NavitrolArrayLimit AND StatusBusy, Socket := TcpSocket, SetRelease := SetNavitrolSpeedLimit, ArrayIndex := SpeedArray);
IF TxMessage3028.Done THEN Navitrol_SpeedUpdate := FALSE; END_IF;
(* Rung 8: Message 3202: Set target detection ControlModeLift *)
TxMessage3032(Enable := TCPReady AND SendTargetDetectionSettings AND StatusBusy, Socket := TcpSocket, Data := PalletDetectionSettings);
IF TxMessage3032.Done THEN SendTargetDetectionSettings := FALSE; END_IF;

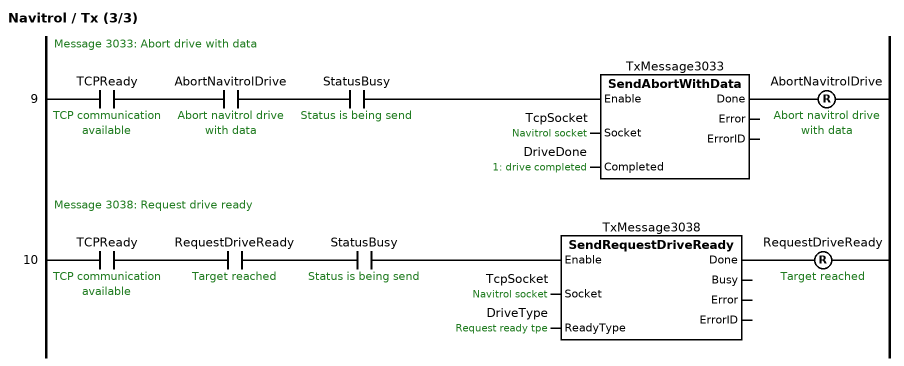
(* Rung 9: Message 3033: Abort drive with data *)
TxMessage3033(Enable := TCPReady AND AbortNavitrolDrive AND StatusBusy, Socket := TcpSocket, Completed := DriveDone);
IF TxMessage3033.Done THEN AbortNavitrolDrive := FALSE; END_IF;
(* Rung 10: Message 3038: Request drive ready *)
TxMessage3038(Enable := TCPReady AND RequestDriveReady AND StatusBusy, Socket := TcpSocket, ReadyType := DriveType);
IF TxMessage3038.Done THEN RequestDriveReady := FALSE; END_IF;

(* Section Rx: ladder, written here as Structured Text *)

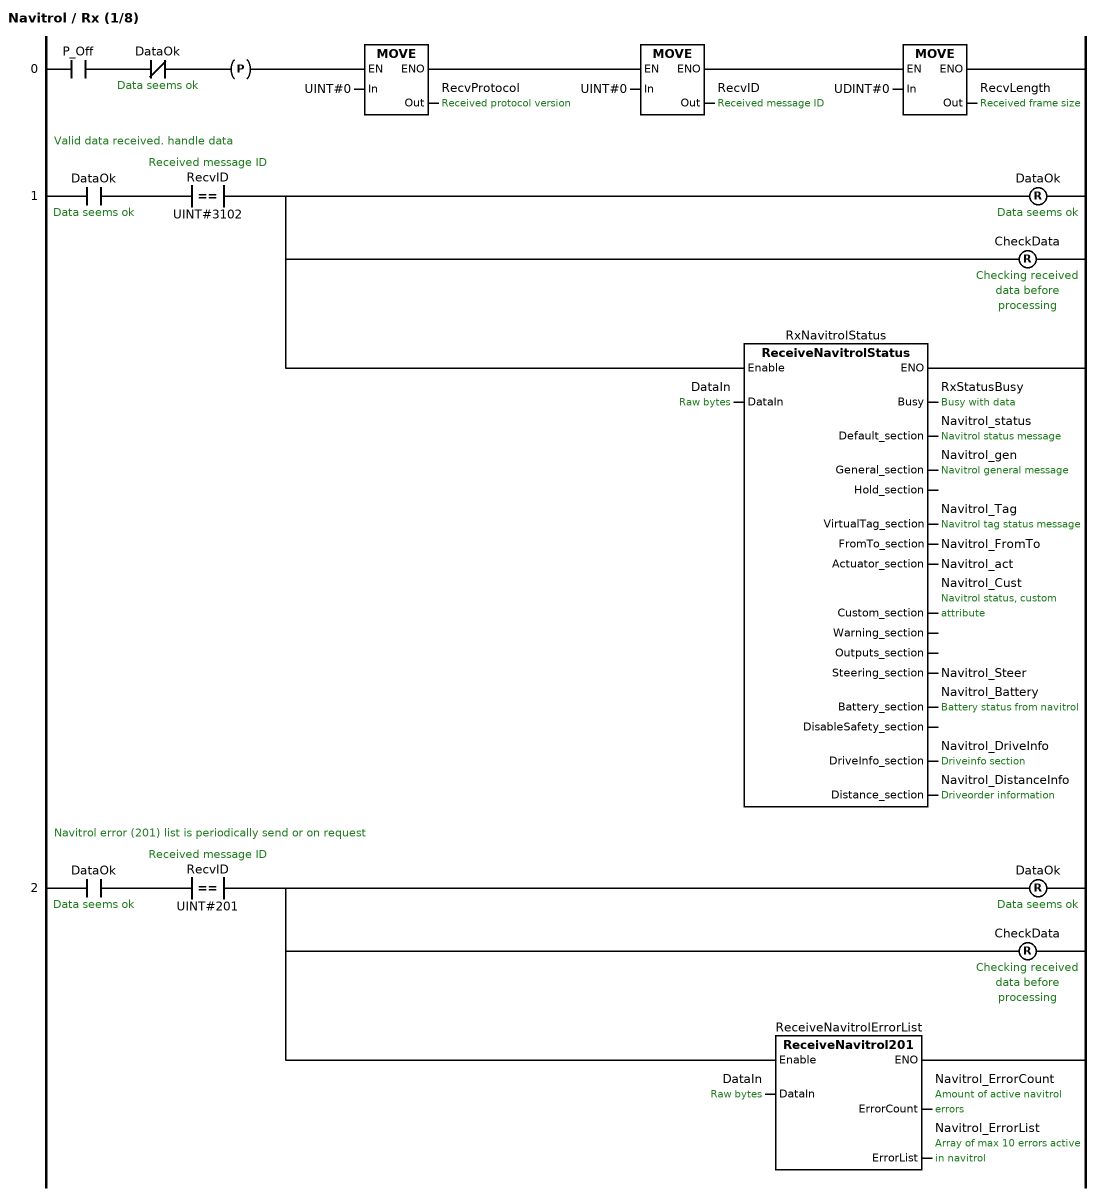
(* Rung 0 *)
_e4(CLK := P_Off AND NOT DataOk);
IF _e4.Q THEN
    RecvProtocol := UINT#0;
    RecvID := UINT#0;
    RecvLength := UDINT#0;
END_IF;
(* Rung 1: Valid data received. handle data *)
_p5 := DataOk AND (RecvID = UINT#3102);
IF _p5 THEN
    DataOk := FALSE;
    CheckData := FALSE;
END_IF;
RxNavitrolStatus(Enable := _p5, DataIn := DataIn, Busy => RxStatusBusy, Default_section => Navitrol_status, General_section => Navitrol_gen, VirtualTag_section => Navitrol_Tag, FromTo_section => Navitrol_FromTo, Actuator_section => Navitrol_act, Custom_section => Navitrol_Cust, Steering_section => Navitrol_Steer, Battery_section => Navitrol_Battery, DriveInfo_section => Navitrol_DriveInfo, Distance_section => Navitrol_DistanceInfo);
(* Rung 2: Navitrol error (201) list is periodically send or on request *)
_p6 := DataOk AND (RecvID = UINT#201);
IF _p6 THEN
    DataOk := FALSE;
    CheckData := FALSE;
END_IF;
ReceiveNavitrolErrorList(Enable := _p6, DataIn := DataIn, ErrorCount => Navitrol_ErrorCount, ErrorList => Navitrol_ErrorList);

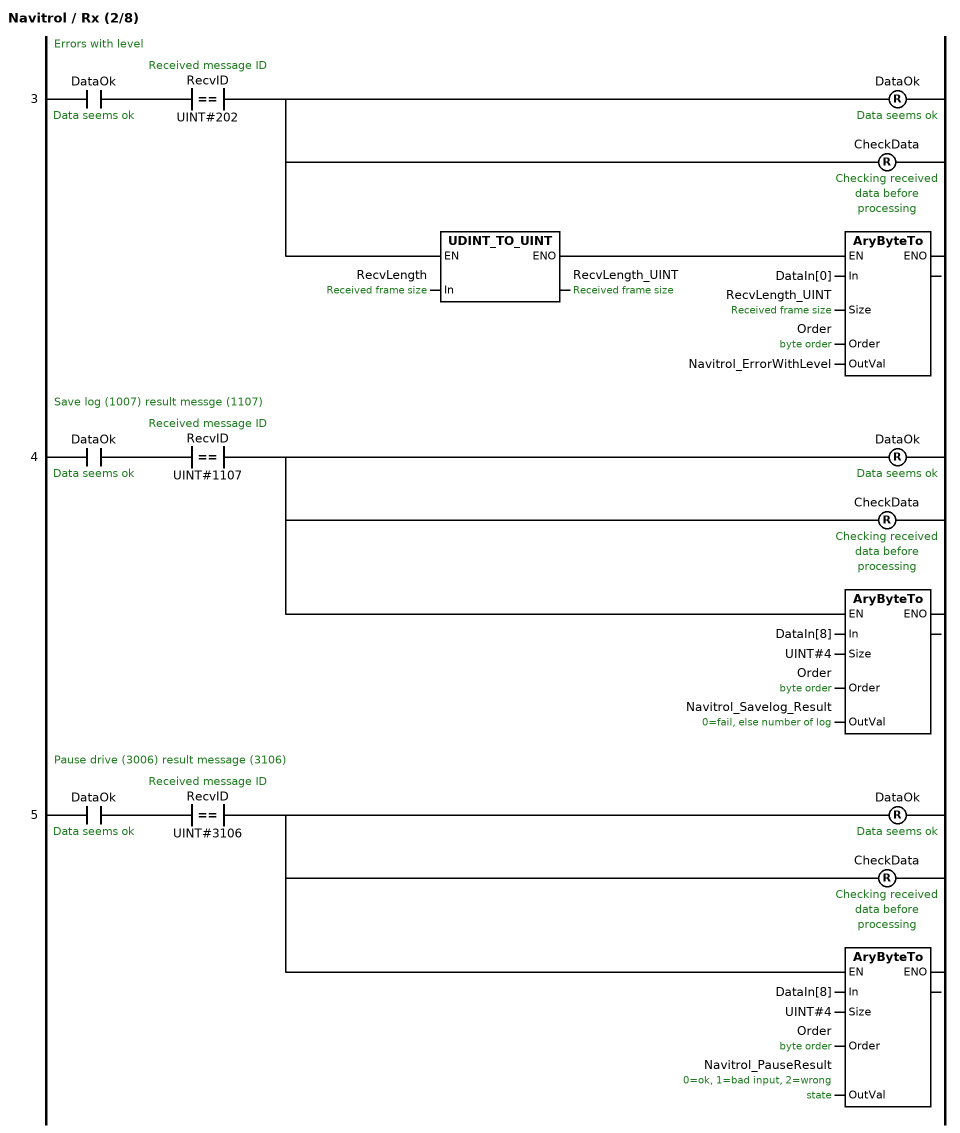
(* Rung 3: Errors with level *)
_p7 := DataOk AND (RecvID = UINT#202);
IF _p7 THEN
    DataOk := FALSE;
    CheckData := FALSE;
    RecvLength_UINT := UDINT_TO_UINT(In := RecvLength);
    AryByteTo(In := DataIn[0], Size := RecvLength_UINT, Order := Order, OutVal := Navitrol_ErrorWithLevel);
END_IF;
(* Rung 4: Save log (1007) result messge (1107) *)
_p8 := DataOk AND (RecvID = UINT#1107);
IF _p8 THEN
    DataOk := FALSE;
    CheckData := FALSE;
    AryByteTo(In := DataIn[8], Size := UINT#4, Order := Order, OutVal := Navitrol_Savelog_Result);
END_IF;
(* Rung 5: Pause drive (3006) result message (3106) *)
_p9 := DataOk AND (RecvID = UINT#3106);
IF _p9 THEN
    DataOk := FALSE;
    CheckData := FALSE;
    AryByteTo(In := DataIn[8], Size := UINT#4, Order := Order, OutVal := Navitrol_PauseResult);
END_IF;

